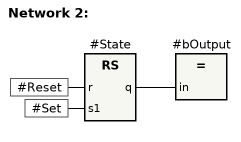
   IF #Reset THEN
       #State := FALSE;   // RS flip-flop
   END_IF;
   IF #Set THEN #State := TRUE; END_IF;
   #bOutput := #State;
END_REGION
END_FUNCTION_BLOCK

FUNCTION_BLOCK "fbLowAlarm"   // FB10, FBD
TITLE = Lightweight version of fbAnalogAlarm with only one limit
{ S7_Optimized_Access := 'TRUE' }
VERSION : 0.1
// stored: AutoNumber true, IsIECCheckEnabled false, IsRetainMemResEnabled false, MemoryReserve 0, SetENOAutomatically false, UDAEnableTagReadback false
   VAR_INPUT
      sValue : "stCalcValue";
      bAckAll : Bool;
      bEnable : Bool;
   END_VAR
   VAR_IN_OUT
      sTag : "stLimitAlarm";
   END_VAR
   VAR
      Alarm : "fbLimitAlarm";
   END_VAR
   VAR CONSTANT
      Low : Bool;
      High : Bool := true;
   END_VAR
BEGIN

REGION Network 1
   // Note that alarm is disabled if CalcValue .bError is set
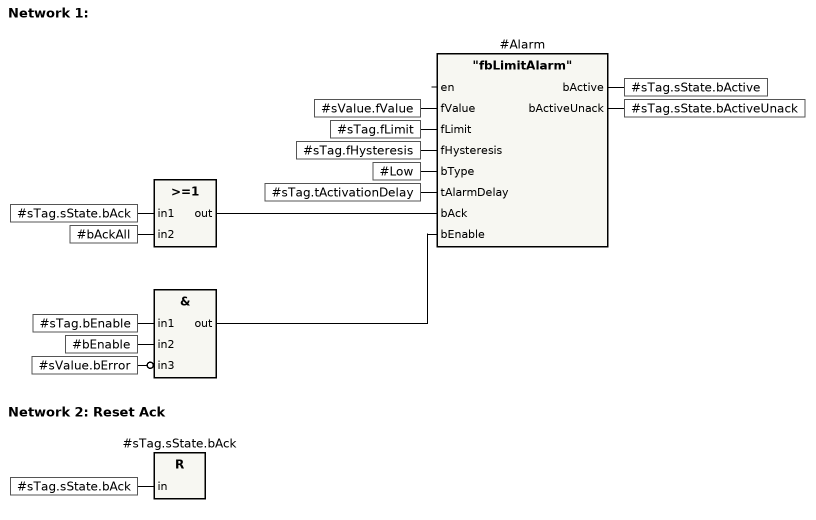
   #Alarm(fValue := #sValue.fValue,   // "fbLimitAlarm"
          fLimit := #sTag.fLimit,
          fHysteresis := #sTag.fHysteresis,
          bType := #Low,
          tAlarmDelay := #sTag.tActivationDelay,
          bAck := #sTag.sState.bAck OR #bAckAll,
          bEnable := #sTag.bEnable AND #bEnable AND NOT #sValue.bError,
          bActive => #sTag.sState.bActive,
          bActiveUnack => #sTag.sState.bActiveUnack);
END_REGION

REGION Network 2: Reset Ack
   IF #sTag.sState.bAck THEN #sTag.sState.bAck := FALSE; END_IF;
END_REGION
END_FUNCTION_BLOCK

FUNCTION_BLOCK "fbDeviationAlarm"   // FB55, FBD
{ S7_Optimized_Access := 'TRUE' }
AUTHOR : Heaten
VERSION : 0.1
// stored: AutoNumber true, IsIECCheckEnabled false, IsRetainMemResEnabled false, MemoryReserve 0, SetENOAutomatically false, UDAEnableTagReadback false
   VAR_INPUT
      sActualValue : "stCalcValue";   // Process value
      fCommandValue : Real;   // Setpoint
      bAckAll : Bool;
      bEnable : Bool;
   END_VAR
   VAR_IN_OUT
      sTag : "stDeviationAlarm";
   END_VAR
   VAR
      Alarm : "fbAlarm";
   END_VAR
   VAR_TEMP
      AlarmCondition : Bool;
   END_VAR
BEGIN

REGION Network 1 (SCL): Alarm condition if measured value ok
   IF #sActualValue.bError = FALSE THEN
       #AlarmCondition := ABS(#sActualValue.fValue - #fCommandValue) > #sTag.fDeviationLimit;
   ELSE
       #AlarmCondition := FALSE;
   END_IF;
END_REGION

REGION Network 2: Alarm with activation delay
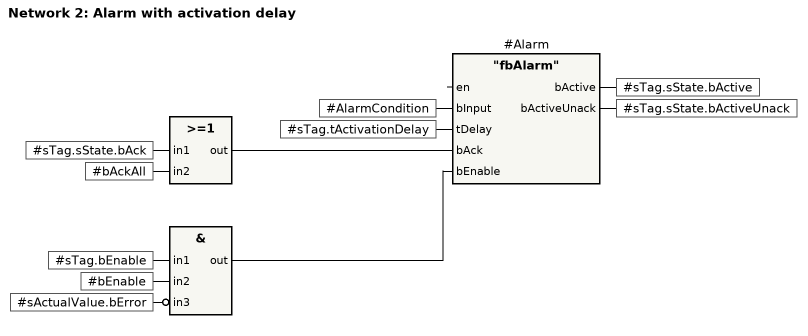
   #Alarm(bInput := #AlarmCondition,   // "fbAlarm"
          tDelay := #sTag.tActivationDelay,
          bAck := #sTag.sState.bAck OR #bAckAll,
          bEnable := #sTag.bEnable AND #bEnable AND NOT #sActualValue.bError,
          bActive => #sTag.sState.bActive,
          bActiveUnack => #sTag.sState.bActiveUnack);
END_REGION
END_FUNCTION_BLOCK

FUNCTION_BLOCK "Regulation"   // FB5, FBD
{ S7_Optimized_Access := 'TRUE' }
VERSION : 0.1
// stored: AutoNumber true, IsIECCheckEnabled true, IsRetainMemResEnabled false, MemoryReserve 10, SetENOAutomatically false, UDAEnableTagReadback false
   VAR
      ExpValveCurrentPressureLimitation : Bool;
      enEmergencyStop { ExternalAccessible := 'False'; ExternalVisible := 'False'; ExternalWritable := 'False'} : Bool;
      CPCPumpRequestFromCPC { ExternalAccessible := 'False'; ExternalVisible := 'False'; ExternalWritable := 'False'} : Bool;   // Crankcase Pressure Control wants to run CPC pump
      CPCPumpRequestFromPurge { ExternalAccessible := 'False'; ExternalVisible := 'False'; ExternalWritable := 'False'} : Bool;   // Do compressor manifold purge
      ExpValveCurrentPressureTarged : Real;
      PerformanceControl_PerformanceRate : Real;
      PerformanceControl { ExternalAccessible := 'False'; ExternalVisible := 'False'; ExternalWritable := 'False'; S7_SetPoint := 'True'} : "PerformanceControl";   // Compressor setpoint
      SuperheatControl { ExternalAccessible := 'False'; ExternalVisible := 'False'; ExternalWritable := 'False'; S7_SetPoint := 'True'} : "SuperheatControl";   // Superheat setpoint
      PinchControl { ExternalAccessible := 'False'; ExternalVisible := 'False'; ExternalWritable := 'False'; S7_SetPoint := 'True'} : "PinchControl";
      CrankcaseOilHeating { ExternalAccessible := 'False'; ExternalVisible := 'False'; ExternalWritable := 'False'; S7_SetPoint := 'True'} : "OilHeating";
      MotorSpeedControl { ExternalAccessible := 'False'; ExternalVisible := 'False'; ExternalWritable := 'False'; S7_SetPoint := 'True'} : "MotorControl";
      SafetyRelay { ExternalAccessible := 'False'; ExternalVisible := 'False'; ExternalWritable := 'False'; S7_SetPoint := 'True'} : "fbSafetyRelay";
      CabinetTemperature { ExternalAccessible := 'False'; ExternalVisible := 'False'; ExternalWritable := 'False'; S7_SetPoint := 'True'} : "fbTemperatureController2";
      ContainerVentilation { ExternalAccessible := 'False'; ExternalVisible := 'False'; ExternalWritable := 'False'; S7_SetPoint := 'True'} : "fbPI_Regulator";
      CrankcasePressureControl { ExternalAccessible := 'False'; ExternalVisible := 'False'; ExternalWritable := 'False'; S7_SetPoint := 'True'} : "CrankcasePressureControl";
      OilSeparator { ExternalAccessible := 'False'; ExternalVisible := 'False'; ExternalWritable := 'False'; S7_SetPoint := 'True'} : "OilSeparator";
      ShaftSealCartridge { ExternalAccessible := 'False'; ExternalVisible := 'False'; ExternalWritable := 'False'; S7_SetPoint := 'True'} : "ShaftSealCartridge";
      LubricationPriming { ExternalAccessible := 'False'; ExternalVisible := 'False'; ExternalWritable := 'False'; S7_SetPoint := 'True'} : "LubricationPriming";
      ValveControl { ExternalAccessible := 'False'; ExternalVisible := 'False'; ExternalWritable := 'False'; S7_SetPoint := 'True'} : "ValveControl";
      PurgeControl { ExternalAccessible := 'False'; ExternalVisible := 'False'; ExternalWritable := 'False'; S7_SetPoint := 'True'} : "fbPurgeControl";
      FilterDryer { S7_SetPoint := 'True'} : "fbFilterDryer";
      OilRecovery { S7_SetPoint := 'True'} : "fbOilRecovery";
      RecuperatorBypass { S7_SetPoint := 'True'} : "fbNullRegulator";
      HeatSourceCycle { S7_SetPoint := 'True'} : "fbTrackingRegulator";
      HeatSourceCyclePIP { S7_SetPoint := 'True'} : "fbPIP_Regulator";
      HeatboosterSetpointPrev { ExternalAccessible := 'False'; ExternalVisible := 'False'; ExternalWritable := 'False'} : Real;   // TEST
      HeatSinkSetpointPrev { ExternalAccessible := 'False'; ExternalVisible := 'False'; ExternalWritable := 'False'} : Real;   // TEST
      HeatSourceSetpointPrev { ExternalAccessible := 'False'; ExternalVisible := 'False'; ExternalWritable := 'False'} : Real;   // TEST
      VariableSetpointPrev { ExternalAccessible := 'False'; ExternalVisible := 'False'; ExternalWritable := 'False'} : Real;
      RegulationTarget { ExternalAccessible := 'False'; ExternalVisible := 'False'; ExternalWritable := 'False'} : Int;   // TEST
      epHeatSinkControlActive { ExternalAccessible := 'False'; ExternalVisible := 'False'; ExternalWritable := 'False'} : Bool;
      epHeatSourceControlActive { ExternalAccessible := 'False'; ExternalVisible := 'False'; ExternalWritable := 'False'} : Bool;
      epVariableControlActive { ExternalAccessible := 'False'; ExternalVisible := 'False'; ExternalWritable := 'False'} : Bool;
      TEST1 : Bool;
   END_VAR
   VAR_TEMP
      AdditionalSuperHeat : Real;
      PerformanceSetpoint : Real;
      AdditionalSuperheatPinch : Real;
   END_VAR
   VAR_TEMP   // added for the SCL form of the ladder/FBD networks
      _w1 : Bool;
   END_VAR
BEGIN

REGION Network 1: Performance control
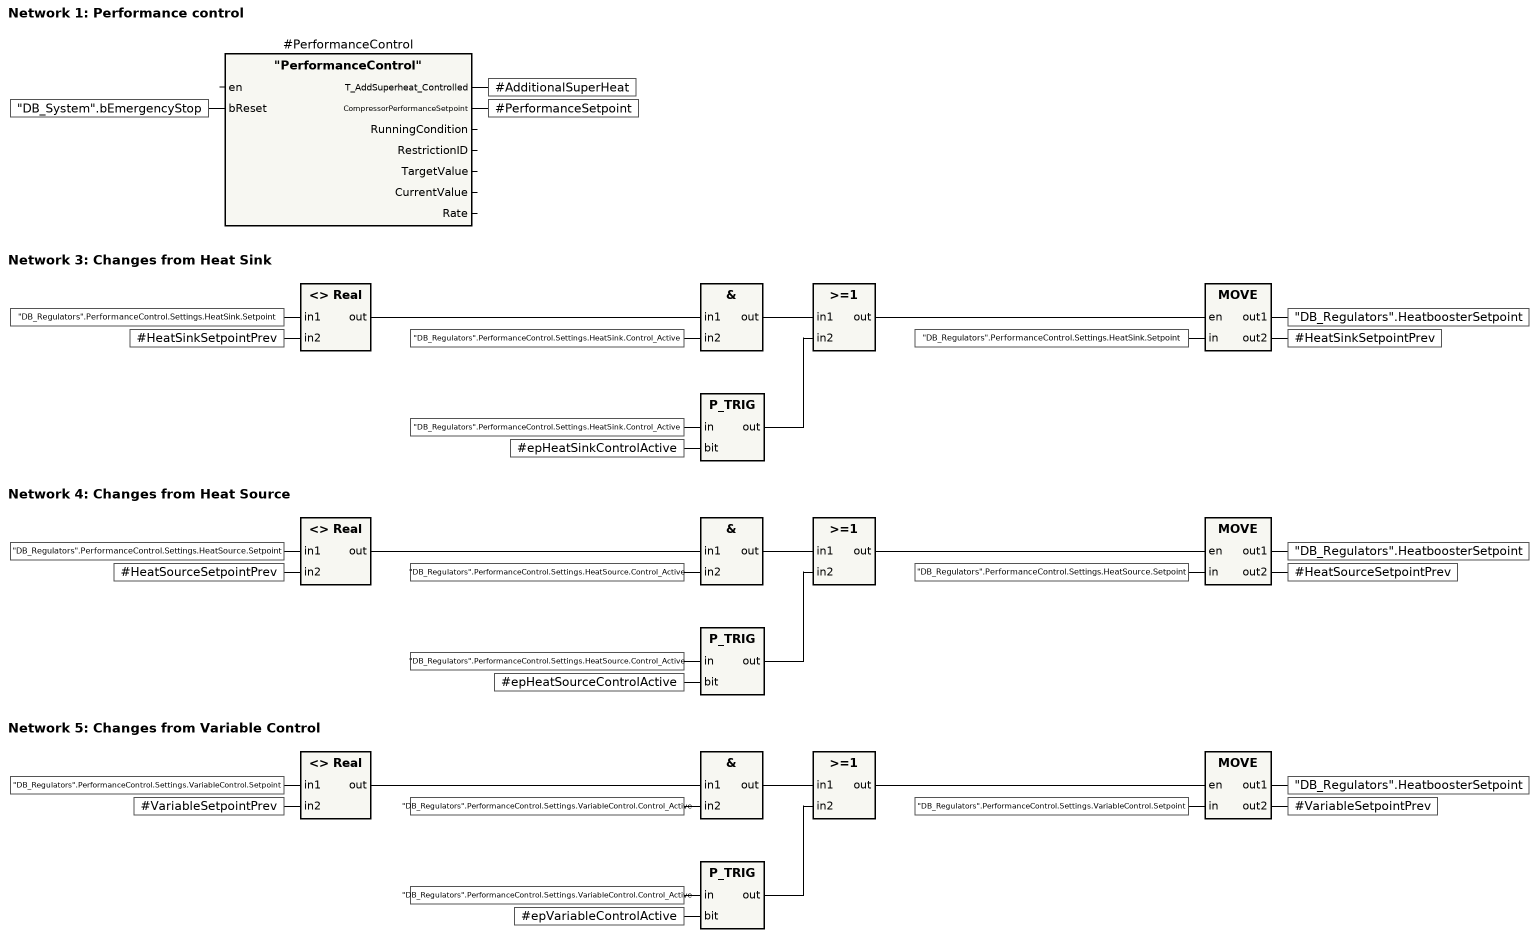
   #PerformanceControl(bReset := "DB_System".bEmergencyStop,   // "PerformanceControl"
                       T_AddSuperheat_Controlled => #AdditionalSuperHeat,
                       CompressorPerformanceSetpoint => #PerformanceSetpoint);
END_REGION

REGION Network 2 (SCL): Performance rate
   // Used in HMI only
   IF "DB_State".State."5_Warmup" OR "DB_State".State."6_Running" AND #PerformanceControl.RunningCondition = TRUE THEN
       #PerformanceControl_PerformanceRate := #MotorSpeedControl.NEngineSetpoint / 15 - #AdditionalSuperHeat / 50 * 30;
   ELSE
       #PerformanceControl_PerformanceRate := 0;
   END_IF;
END_REGION

REGION Network 3: Changes from Heat Sink
   // Propagate setpoint when controller is first activated, or if active and setpoint is changed
   #_w1 := "DB_Regulators".PerformanceControl.Settings.HeatSink.Control_Active AND NOT #epHeatSinkControlActive;   // rising edge
   #epHeatSinkControlActive := "DB_Regulators".PerformanceControl.Settings.HeatSink.Control_Active;
   IF (("DB_Regulators".PerformanceControl.Settings.HeatSink.Setpoint <> #HeatSinkSetpointPrev) AND "DB_Regulators".PerformanceControl.Settings.HeatSink.Control_Active) OR #_w1 THEN
       "DB_Regulators".HeatboosterSetpoint := "DB_Regulators".PerformanceControl.Settings.HeatSink.Setpoint;
       #HeatSinkSetpointPrev := "DB_Regulators".PerformanceControl.Settings.HeatSink.Setpoint;
   END_IF;
END_REGION

REGION Network 4: Changes from Heat Source
   // Propagate setpoint when controller is first activated, or if active and setpoint is changed
   #_w1 := "DB_Regulators".PerformanceControl.Settings.HeatSource.Control_Active AND NOT #epHeatSourceControlActive;   // rising edge
   #epHeatSourceControlActive := "DB_Regulators".PerformanceControl.Settings.HeatSource.Control_Active;
   IF (("DB_Regulators".PerformanceControl.Settings.HeatSource.Setpoint <> #HeatSourceSetpointPrev) AND "DB_Regulators".PerformanceControl.Settings.HeatSource.Control_Active) OR #_w1 THEN
       "DB_Regulators".HeatboosterSetpoint := "DB_Regulators".PerformanceControl.Settings.HeatSource.Setpoint;
       #HeatSourceSetpointPrev := "DB_Regulators".PerformanceControl.Settings.HeatSource.Setpoint;
   END_IF;
END_REGION

REGION Network 5: Changes from Variable Control
   // Propagate setpoint when controller is first activated, or if active and setpoint is changed
   #_w1 := "DB_Regulators".PerformanceControl.Settings.VariableControl.Control_Active AND NOT #epVariableControlActive;   // rising edge
   #epVariableControlActive := "DB_Regulators".PerformanceControl.Settings.VariableControl.Control_Active;
   IF (("DB_Regulators".PerformanceControl.Settings.VariableControl.Setpoint <> #VariableSetpointPrev) AND "DB_Regulators".PerformanceControl.Settings.VariableControl.Control_Active) OR #_w1 THEN
       "DB_Regulators".HeatboosterSetpoint := "DB_Regulators".PerformanceControl.Settings.VariableControl.Setpoint;
       #VariableSetpointPrev := "DB_Regulators".PerformanceControl.Settings.VariableControl.Setpoint;
   END_IF;
END_REGION

REGION Network 6 (SCL): Regulation target
   // No, I didn't suddenly develop a brain hemorrage, this mess here is on purpose:
   // 1. It is a sequence of separate IFs as it mirrors the logic in PerformanceControl
   // 2. It is tempting to re-use Restriction ID, but this can take on values other than the ones here, which we want to avoid. So the value has to be reconstructed.
   // Figure out which target is active
   "DB_Regulators".RegulationTarget := 0;  // in case none of the regulators are active, none of the IFs fire...
   IF "DB_Regulators".PerformanceControl.Settings.HeatSink.Control_Active THEN
       IF "DB_Regulators".PerformanceControl.Settings.HeatSink.UseFeedFlow THEN
           "DB_Regulators".RegulationTarget := 2;
       ELSE
           "DB_Regulators".RegulationTarget := 1;
       END_IF;
   END_IF;

   IF "DB_Regulators".PerformanceControl.Settings.HeatSource.Control_Active THEN
       IF "DB_Regulators".PerformanceControl.Settings.HeatSource.UseFeedFlow THEN
           "DB_Regulators".RegulationTarget := 4;
       ELSE
           "DB_Regulators".RegulationTarget := 3;
       END_IF;
   END_IF;

   IF "DB_Regulators".PerformanceControl.Settings.VariableControl.Control_Active AND "DB_Regulators".PerformanceControl.Settings.VariableControl.ReferenceID > 0 THEN
       "DB_Regulators".RegulationTarget := 6;
   END_IF;
END_REGION

REGION Network 7: Changes from DB_Regulators
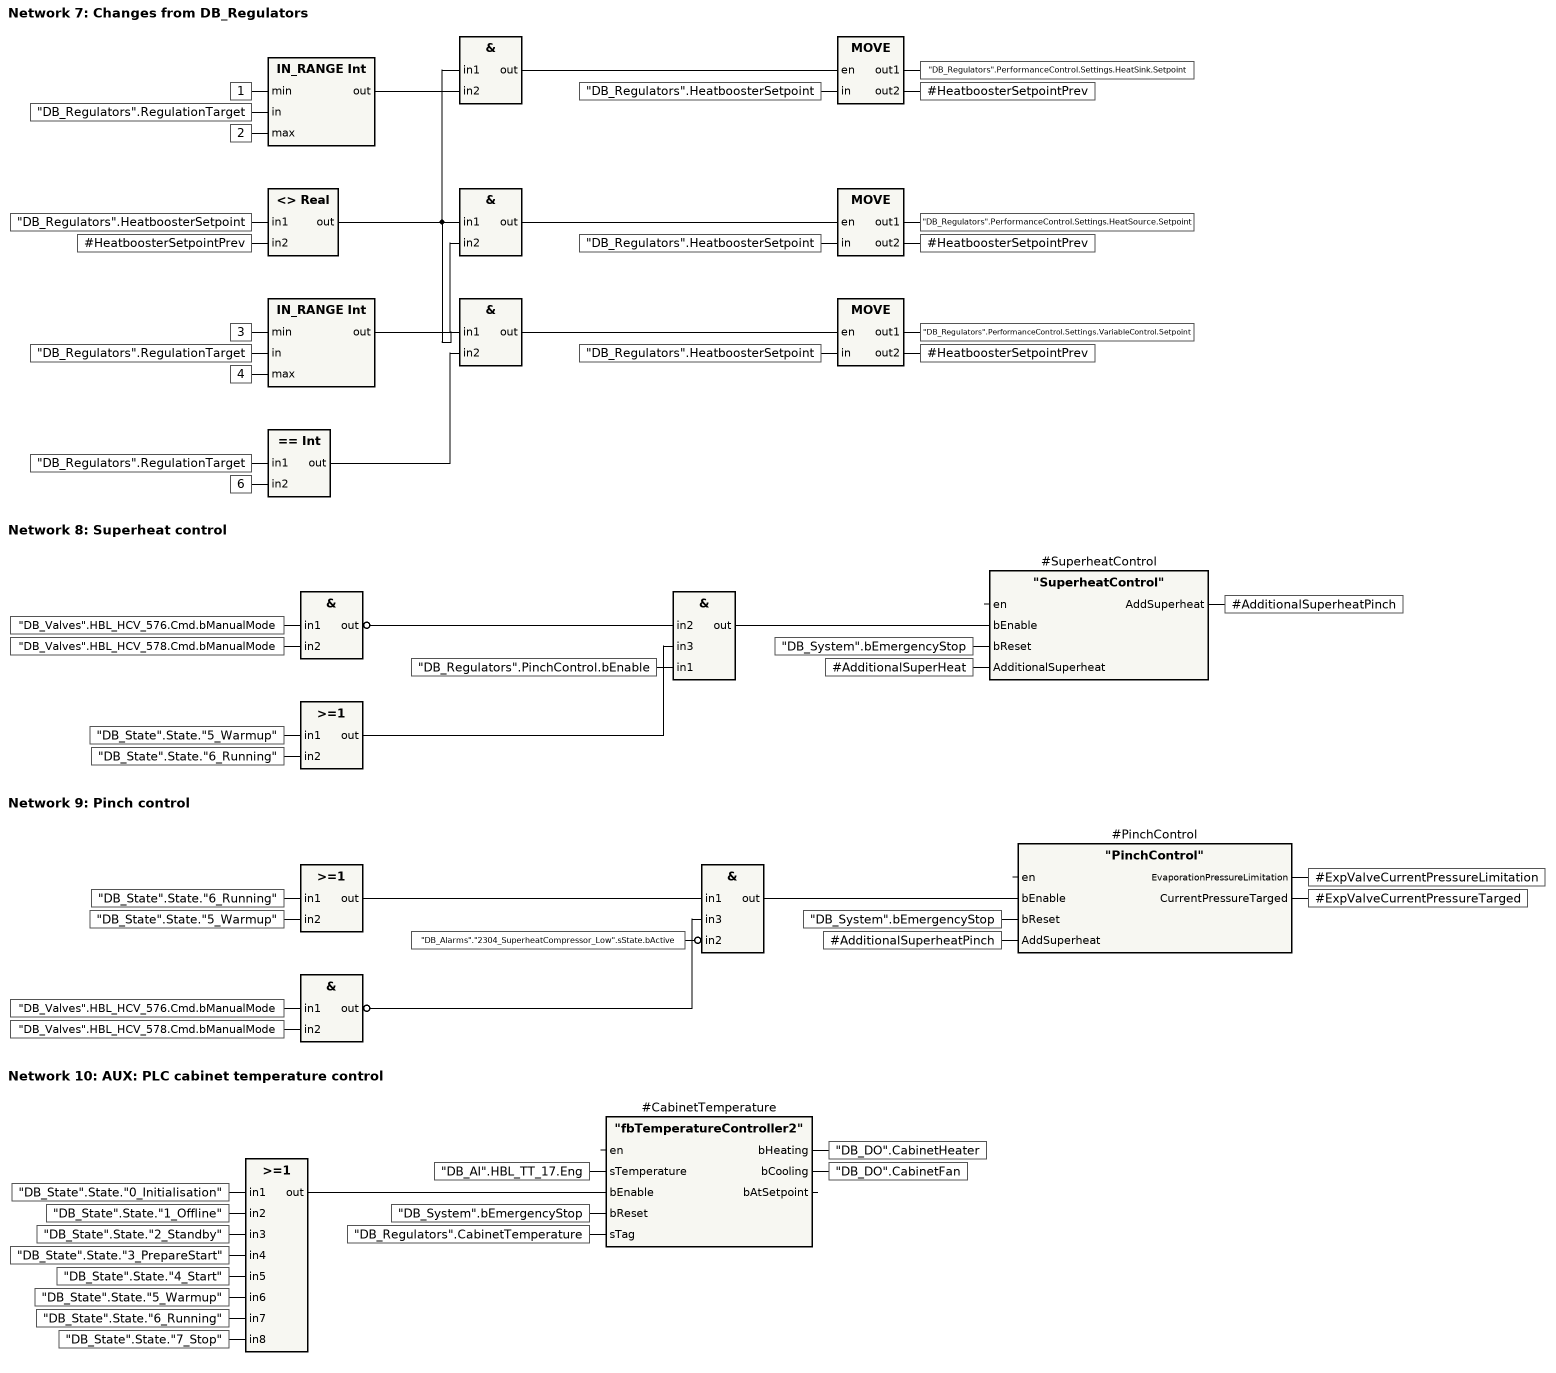
   #_w1 := "DB_Regulators".HeatboosterSetpoint <> #HeatboosterSetpointPrev;
   IF #_w1 AND (1 <= "DB_Regulators".RegulationTarget) AND ("DB_Regulators".RegulationTarget <= 2) THEN
       "DB_Regulators".PerformanceControl.Settings.HeatSink.Setpoint := "DB_Regulators".HeatboosterSetpoint;
       #HeatboosterSetpointPrev := "DB_Regulators".HeatboosterSetpoint;
   END_IF;
   IF #_w1 AND (3 <= "DB_Regulators".RegulationTarget) AND ("DB_Regulators".RegulationTarget <= 4) THEN
       "DB_Regulators".PerformanceControl.Settings.HeatSource.Setpoint := "DB_Regulators".HeatboosterSetpoint;
       #HeatboosterSetpointPrev := "DB_Regulators".HeatboosterSetpoint;
   END_IF;
   IF #_w1 AND ("DB_Regulators".RegulationTarget = 6) THEN
       "DB_Regulators".PerformanceControl.Settings.VariableControl.Setpoint := "DB_Regulators".HeatboosterSetpoint;
       #HeatboosterSetpointPrev := "DB_Regulators".HeatboosterSetpoint;
   END_IF;
END_REGION

REGION Network 8: Superheat control
   #SuperheatControl(bEnable := NOT ("DB_Valves".HBL_HCV_576.Cmd.bManualMode AND "DB_Valves".HBL_HCV_578.Cmd.bManualMode) AND ("DB_State".State."5_Warmup" OR "DB_State".State."6_Running") AND "DB_Regulators".PinchControl.bEnable,   // "SuperheatControl"
                     bReset := "DB_System".bEmergencyStop,
                     AdditionalSuperheat := #AdditionalSuperHeat,
                     AddSuperheat => #AdditionalSuperheatPinch);
END_REGION

REGION Network 9: Pinch control
   #PinchControl(bEnable := ("DB_State".State."6_Running" OR "DB_State".State."5_Warmup") AND NOT ("DB_Valves".HBL_HCV_576.Cmd.bManualMode AND "DB_Valves".HBL_HCV_578.Cmd.bManualMode) AND NOT "DB_Alarms"."2304_SuperheatCompressor_Low".sState.bActive,   // "PinchControl"
                 bReset := "DB_System".bEmergencyStop,
                 AddSuperheat := #AdditionalSuperheatPinch,
                 EvaporationPressureLimitation => #ExpValveCurrentPressureLimitation,
                 CurrentPressureTarged => #ExpValveCurrentPressureTarged);
END_REGION

REGION Network 10: AUX: PLC cabinet temperature control
   // Runs all the time, as the cabinet is running all the time...
   #CabinetTemperature(sTemperature := "DB_AI".HBL_TT_17.Eng,   // "fbTemperatureController2"
                       bEnable := "DB_State".State."0_Initialisation" OR "DB_State".State."1_Offline" OR "DB_State".State."2_Standby" OR "DB_State".State."3_PrepareStart" OR "DB_State".State."4_Start" OR "DB_State".State."5_Warmup" OR "DB_State".State."6_Running" OR "DB_State".State."7_Stop",
                       bReset := "DB_System".bEmergencyStop,
                       sTag := "DB_Regulators".CabinetTemperature,
                       bHeating => "DB_DO".CabinetHeater,
                       bCooling => "DB_DO".CabinetFan);
END_REGION

REGION Network 11: AUX: Crankcase oil heater control
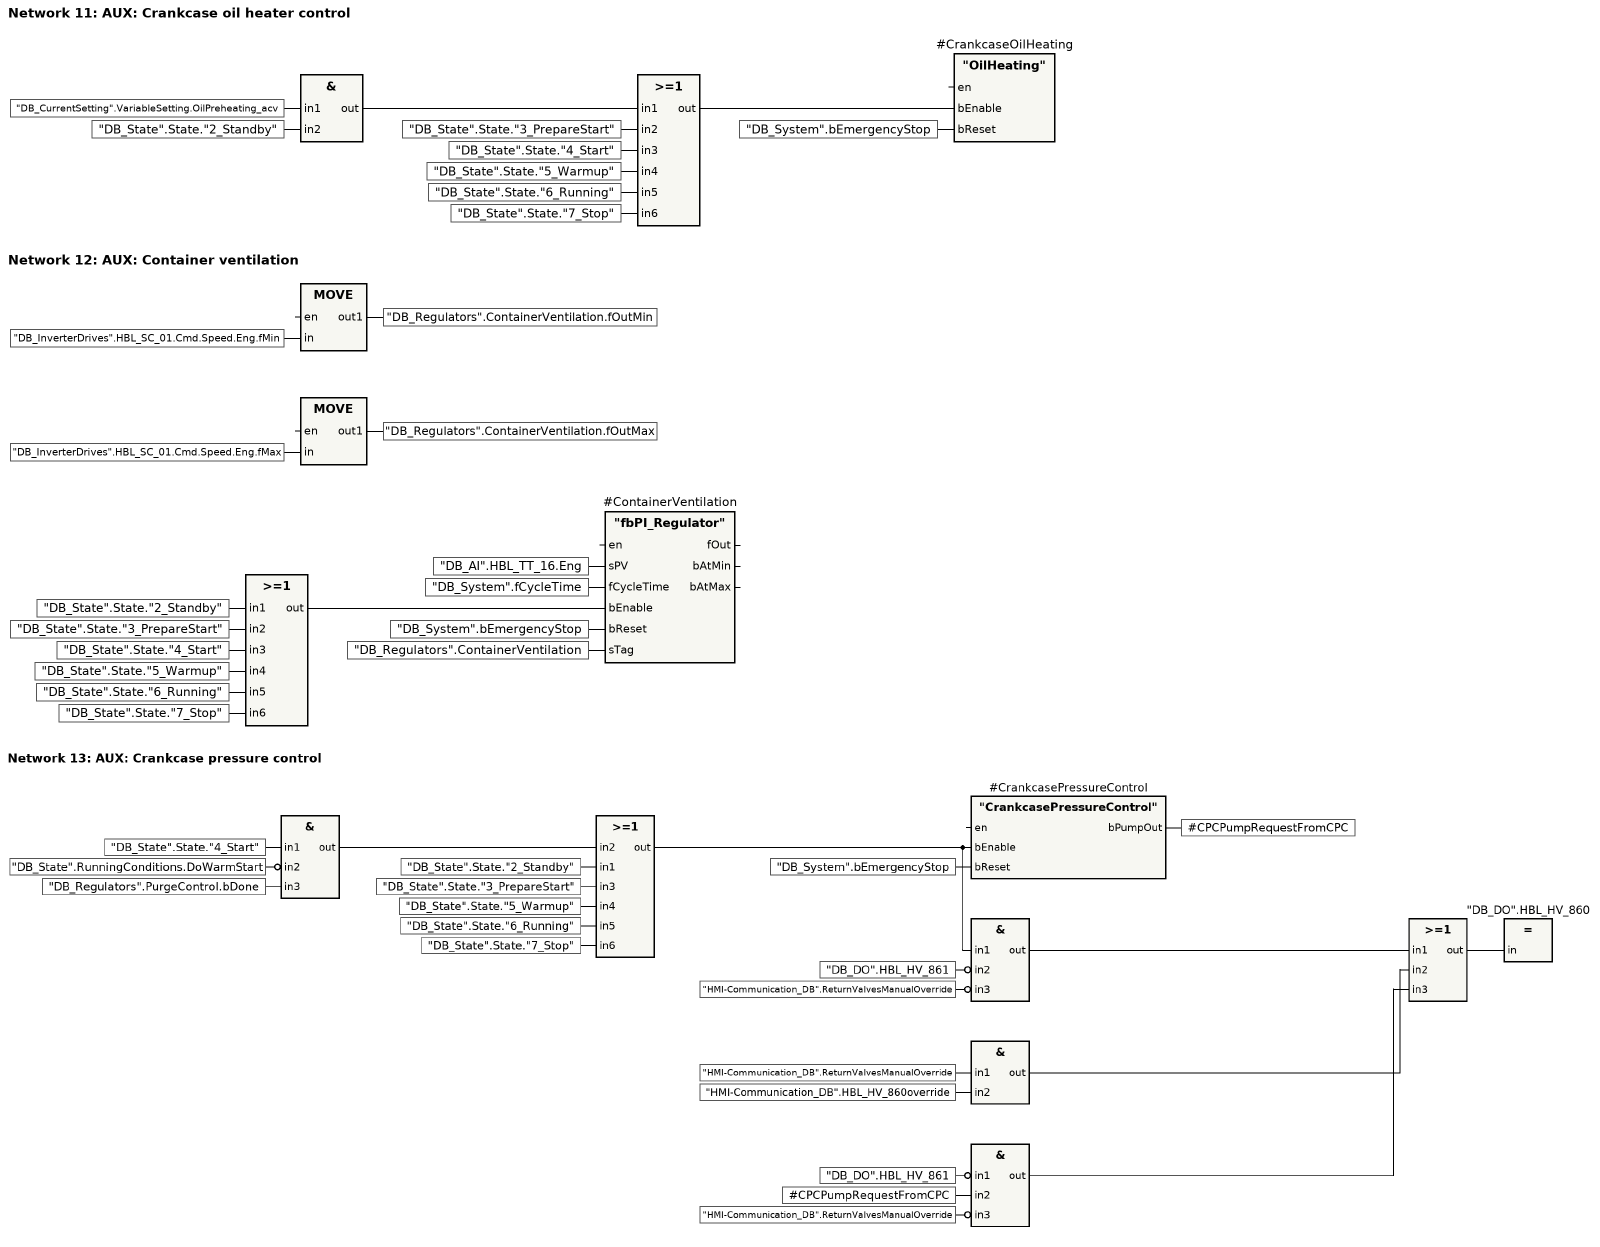
   #CrankcaseOilHeating(bEnable := ("DB_CurrentSetting".VariableSetting.OilPreheating_acv AND "DB_State".State."2_Standby") OR "DB_State".State."3_PrepareStart" OR "DB_State".State."4_Start" OR "DB_State".State."5_Warmup" OR "DB_State".State."6_Running" OR "DB_State".State."7_Stop",   // "OilHeating"
                        bReset := "DB_System".bEmergencyStop);
END_REGION

REGION Network 12: AUX: Container ventilation
   // Manually copy the actuator min & max to the regulator min & max. This is not automatically true for all regulators
   // ##FIX: Hack the start signal, ugliness alert
   "DB_Regulators".ContainerVentilation.fOutMin := "DB_InverterDrives".HBL_SC_01.Cmd.Speed.Eng.fMin;
   "DB_Regulators".ContainerVentilation.fOutMax := "DB_InverterDrives".HBL_SC_01.Cmd.Speed.Eng.fMax;
   #ContainerVentilation(sPV := "DB_AI".HBL_TT_16.Eng,   // "fbPI_Regulator"
                         fCycleTime := "DB_System".fCycleTime,
                         bEnable := "DB_State".State."2_Standby" OR "DB_State".State."3_PrepareStart" OR "DB_State".State."4_Start" OR "DB_State".State."5_Warmup" OR "DB_State".State."6_Running" OR "DB_State".State."7_Stop",
                         bReset := "DB_System".bEmergencyStop,
                         sTag := "DB_Regulators".ContainerVentilation);
END_REGION

REGION Network 13: AUX: Crankcase pressure control
   // Disable the controller temporarily in State 4 Start when doing a cold start
   #_w1 := ("DB_State".State."4_Start" AND NOT "DB_State".RunningConditions.DoWarmStart AND "DB_Regulators".PurgeControl.bDone) OR "DB_State".State."2_Standby" OR "DB_State".State."3_PrepareStart" OR "DB_State".State."5_Warmup" OR "DB_State".State."6_Running" OR "DB_State".State."7_Stop";
   #CrankcasePressureControl(bEnable := #_w1,   // "CrankcasePressureControl"
                           bReset := "DB_System".bEmergencyStop,
                           bPumpOut => #CPCPumpRequestFromCPC);
   "DB_DO".HBL_HV_860 := (#_w1 AND NOT "DB_DO".HBL_HV_861 AND NOT "HMI-Communication_DB".ReturnValvesManualOverride) OR ("HMI-Communication_DB".ReturnValvesManualOverride AND "HMI-Communication_DB".HBL_HV_860override) OR (NOT "DB_DO".HBL_HV_861 AND #CPCPumpRequestFromCPC AND NOT "HMI-Communication_DB".ReturnValvesManualOverride);
END_REGION

REGION Network 14: AUX: Oil separator level control
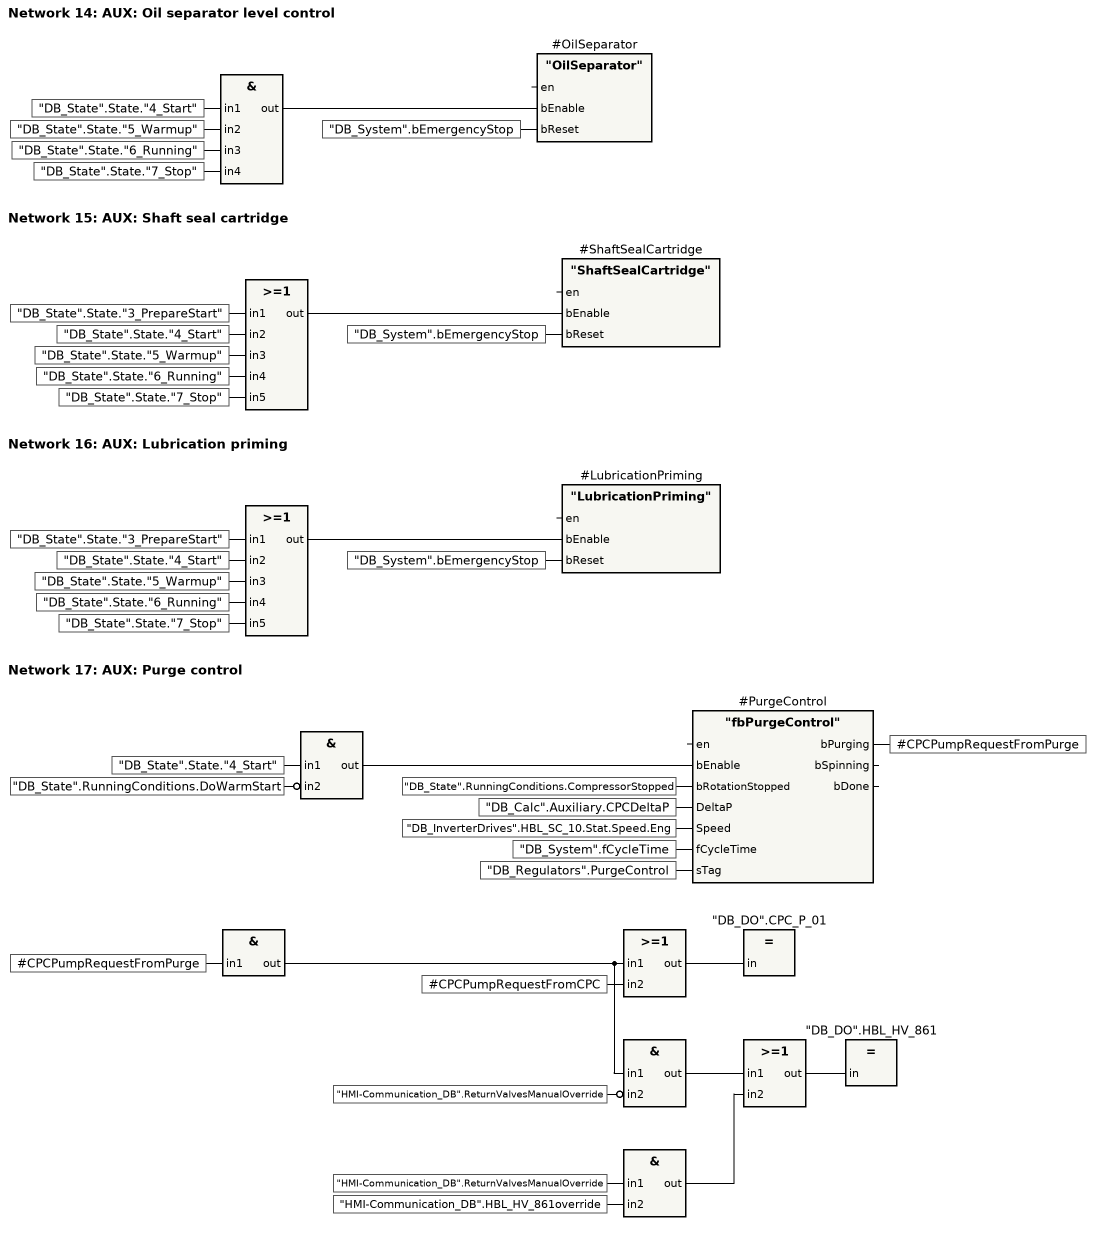
   #OilSeparator(bEnable := "DB_State".State."4_Start" AND "DB_State".State."5_Warmup" AND "DB_State".State."6_Running" AND "DB_State".State."7_Stop",   // "OilSeparator"
                 bReset := "DB_System".bEmergencyStop);
END_REGION

REGION Network 15: AUX: Shaft seal cartridge
   #ShaftSealCartridge(bEnable := "DB_State".State."3_PrepareStart" OR "DB_State".State."4_Start" OR "DB_State".State."5_Warmup" OR "DB_State".State."6_Running" OR "DB_State".State."7_Stop",   // "ShaftSealCartridge"
                       bReset := "DB_System".bEmergencyStop);
END_REGION

REGION Network 16: AUX: Lubrication priming
   #LubricationPriming(bEnable := "DB_State".State."3_PrepareStart" OR "DB_State".State."4_Start" OR "DB_State".State."5_Warmup" OR "DB_State".State."6_Running" OR "DB_State".State."7_Stop",   // "LubricationPriming"
                       bReset := "DB_System".bEmergencyStop);
END_REGION

REGION Network 17: AUX: Purge control
   // Note: HBL-XV-05 takes priority over HBL-XV-04
   #PurgeControl(bEnable := "DB_State".State."4_Start" AND NOT "DB_State".RunningConditions.DoWarmStart,   // "fbPurgeControl"
                 bRotationStopped := "DB_State".RunningConditions.CompressorStopped,
                 DeltaP := "DB_Calc".Auxiliary.CPCDeltaP,
                 Speed := "DB_InverterDrives".HBL_SC_10.Stat.Speed.Eng,
                 fCycleTime := "DB_System".fCycleTime,
                 sTag := "DB_Regulators".PurgeControl,
                 bPurging => #CPCPumpRequestFromPurge);
   "DB_DO".CPC_P_01 := #CPCPumpRequestFromPurge OR #CPCPumpRequestFromCPC;
   "DB_DO".HBL_HV_861 := (#CPCPumpRequestFromPurge AND NOT "HMI-Communication_DB".ReturnValvesManualOverride) OR ("HMI-Communication_DB".ReturnValvesManualOverride AND "HMI-Communication_DB".HBL_HV_861override);
END_REGION

REGION Network 18: AUX: Compressor manifold oil return
   // This is still up in the air what this will be
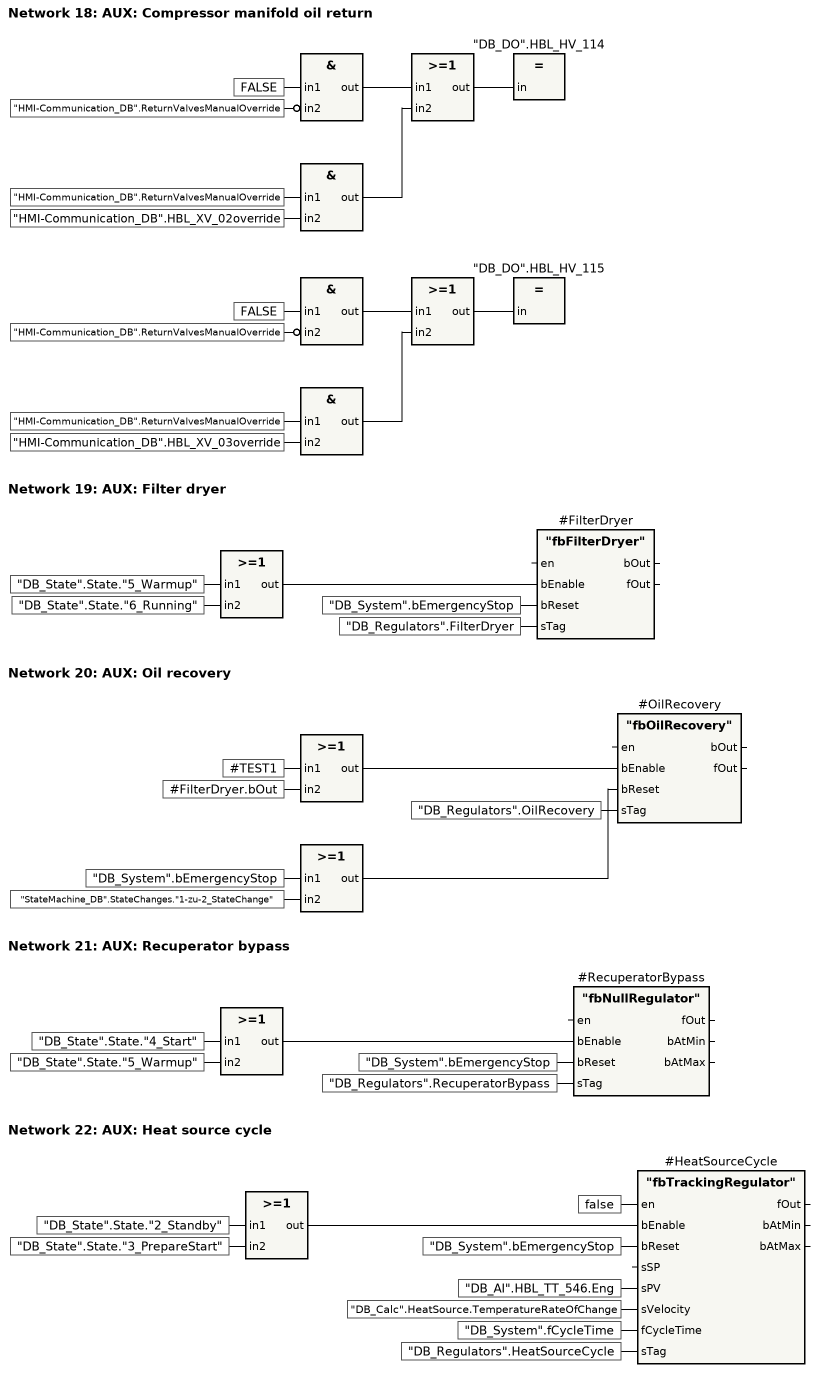
   "DB_DO".HBL_HV_114 := (FALSE AND NOT "HMI-Communication_DB".ReturnValvesManualOverride) OR ("HMI-Communication_DB".ReturnValvesManualOverride AND "HMI-Communication_DB".HBL_XV_02override);
   "DB_DO".HBL_HV_115 := (FALSE AND NOT "HMI-Communication_DB".ReturnValvesManualOverride) OR ("HMI-Communication_DB".ReturnValvesManualOverride AND "HMI-Communication_DB".HBL_XV_03override);
END_REGION

REGION Network 19: AUX: Filter dryer
   #FilterDryer(bEnable := "DB_State".State."5_Warmup" OR "DB_State".State."6_Running",   // "fbFilterDryer"
                bReset := "DB_System".bEmergencyStop,
                sTag := "DB_Regulators".FilterDryer);
END_REGION

REGION Network 20: AUX: Oil recovery
   // Run only when filter dryer is also running
   #OilRecovery(bEnable := #TEST1 OR #FilterDryer.bOut,   // "fbOilRecovery"
                bReset := "DB_System".bEmergencyStop OR "StateMachine_DB".StateChanges."1-zu-2_StateChange",
                sTag := "DB_Regulators".OilRecovery);
END_REGION

REGION Network 21: AUX: Recuperator bypass
   #RecuperatorBypass(bEnable := "DB_State".State."4_Start" OR "DB_State".State."5_Warmup",   // "fbNullRegulator"
                      bReset := "DB_System".bEmergencyStop,
                      sTag := "DB_Regulators".RecuperatorBypass);
END_REGION

REGION Network 22: AUX: Heat source cycle
   IF false THEN
       #HeatSourceCycle(bEnable := "DB_State".State."2_Standby" OR "DB_State".State."3_PrepareStart",   // "fbTrackingRegulator"
                        bReset := "DB_System".bEmergencyStop,
                        sPV := "DB_AI".HBL_TT_546.Eng,
                        sVelocity := "DB_Calc".HeatSource.TemperatureRateOfChange,
                        fCycleTime := "DB_System".fCycleTime,
                        sTag := "DB_Regulators".HeatSourceCycle);
   END_IF;
END_REGION

REGION Network 23: AUX: Heat source cycle PIP
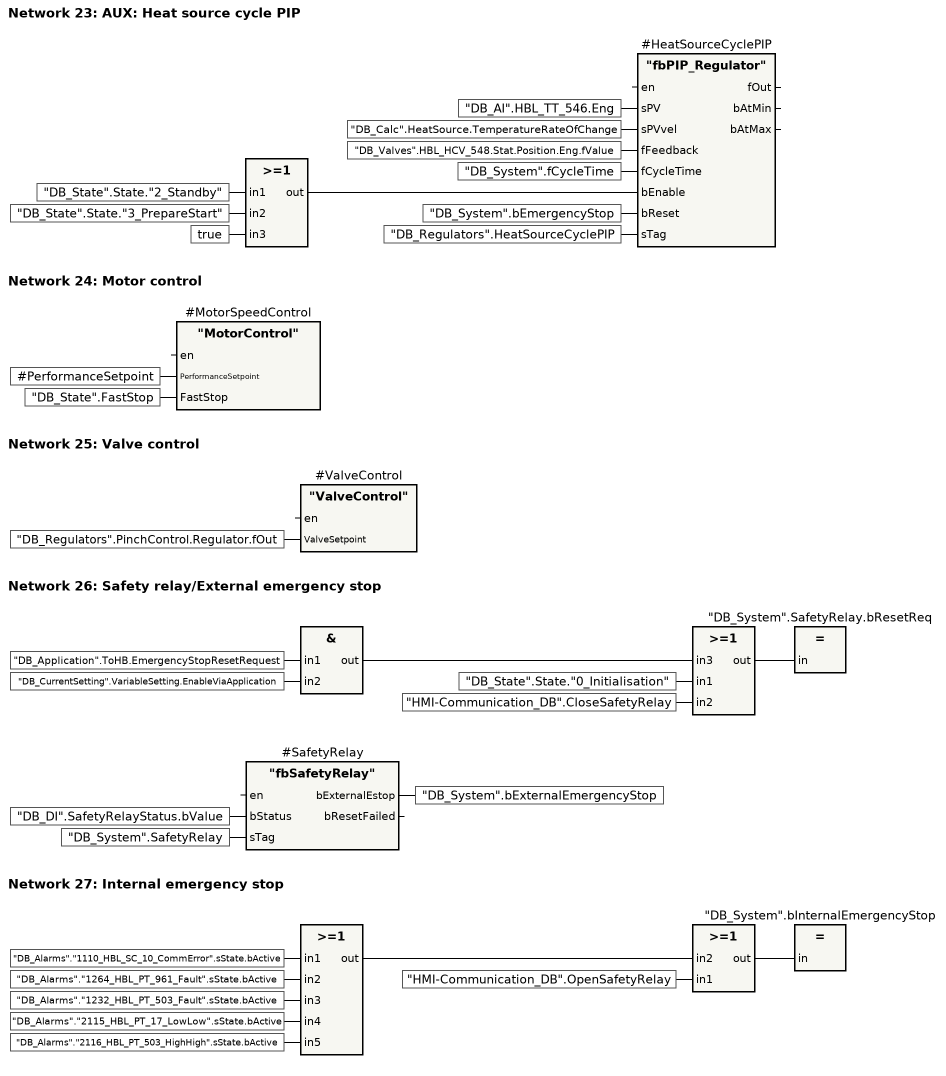
   #HeatSourceCyclePIP(sPV := "DB_AI".HBL_TT_546.Eng,   // "fbPIP_Regulator"
                       sPVvel := "DB_Calc".HeatSource.TemperatureRateOfChange,
                       fFeedback := "DB_Valves".HBL_HCV_548.Stat.Position.Eng.fValue,
                       fCycleTime := "DB_System".fCycleTime,
                       bEnable := "DB_State".State."2_Standby" OR "DB_State".State."3_PrepareStart" OR true,
                       bReset := "DB_System".bEmergencyStop,
                       sTag := "DB_Regulators".HeatSourceCyclePIP);
END_REGION

REGION Network 24: Motor control
   // Note this has to come after all regulators which set the motor speed
   #MotorSpeedControl(PerformanceSetpoint := #PerformanceSetpoint, FastStop := "DB_State".FastStop);   // "MotorControl"
END_REGION

REGION Network 25: Valve control
   #ValveControl(ValveSetpoint := "DB_Regulators".PinchControl.Regulator.fOut);   // "ValveControl"
END_REGION

REGION Network 26: Safety relay/External emergency stop
   "DB_System".SafetyRelay.bResetReq := ("DB_Application".ToHB.EmergencyStopResetRequest AND "DB_CurrentSetting".VariableSetting.EnableViaApplication) OR "DB_State".State."0_Initialisation" OR "HMI-Communication_DB".CloseSafetyRelay;
   #SafetyRelay(bStatus := "DB_DI".SafetyRelayStatus.bValue,   // "fbSafetyRelay"
                sTag := "DB_System".SafetyRelay,
                bExternalEstop => "DB_System".bExternalEmergencyStop);
END_REGION

REGION Network 27: Internal emergency stop
   // The alarms in this list should also be in the Critical alarms list in FB32 AlarmManagement.
   // HBL-PT-17 : lubrication failure, stop compressor (or fault in this sensor)
   // HBL-PT-503: compressor discharge overpressure, stop the compressor (or fault in this sensor)
   // HBL-SC-10: compressor inverter communication loss, no other way to shut it down except by hardwired emergency stop.
   "DB_System".bInternalEmergencyStop := "DB_Alarms"."1110_HBL_SC_10_CommError".sState.bActive OR "DB_Alarms"."1264_HBL_PT_961_Fault".sState.bActive OR "DB_Alarms"."1232_HBL_PT_503_Fault".sState.bActive OR "DB_Alarms"."2115_HBL_PT_17_LowLow".sState.bActive OR "DB_Alarms"."2116_HBL_PT_503_HighHigh".sState.bActive OR "HMI-Communication_DB".OpenSafetyRelay;
END_REGION

REGION Network 28: Emergency stop
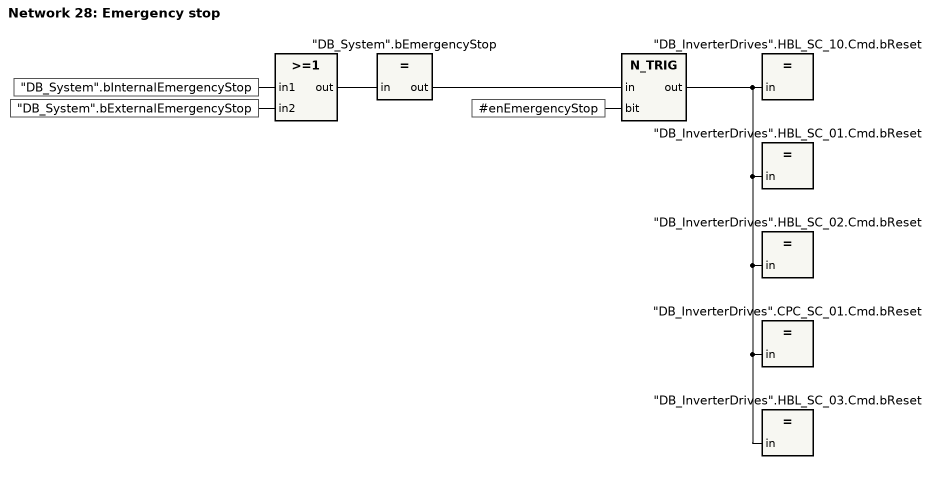
   "DB_System".bEmergencyStop := "DB_System".bInternalEmergencyStop OR "DB_System".bExternalEmergencyStop;
   #_w1 := NOT "DB_System".bEmergencyStop AND #enEmergencyStop;   // falling edge
   #enEmergencyStop := "DB_System".bEmergencyStop;
   "DB_InverterDrives".HBL_SC_10.Cmd.bReset := #_w1;
   "DB_InverterDrives".HBL_SC_01.Cmd.bReset := #_w1;
   "DB_InverterDrives".HBL_SC_02.Cmd.bReset := #_w1;
   "DB_InverterDrives".CPC_SC_01.Cmd.bReset := #_w1;
   "DB_InverterDrives".HBL_SC_03.Cmd.bReset := #_w1;
END_REGION

REGION Network 29: Manual mode warning
   // One or more regulators or actuators is in manual mode.
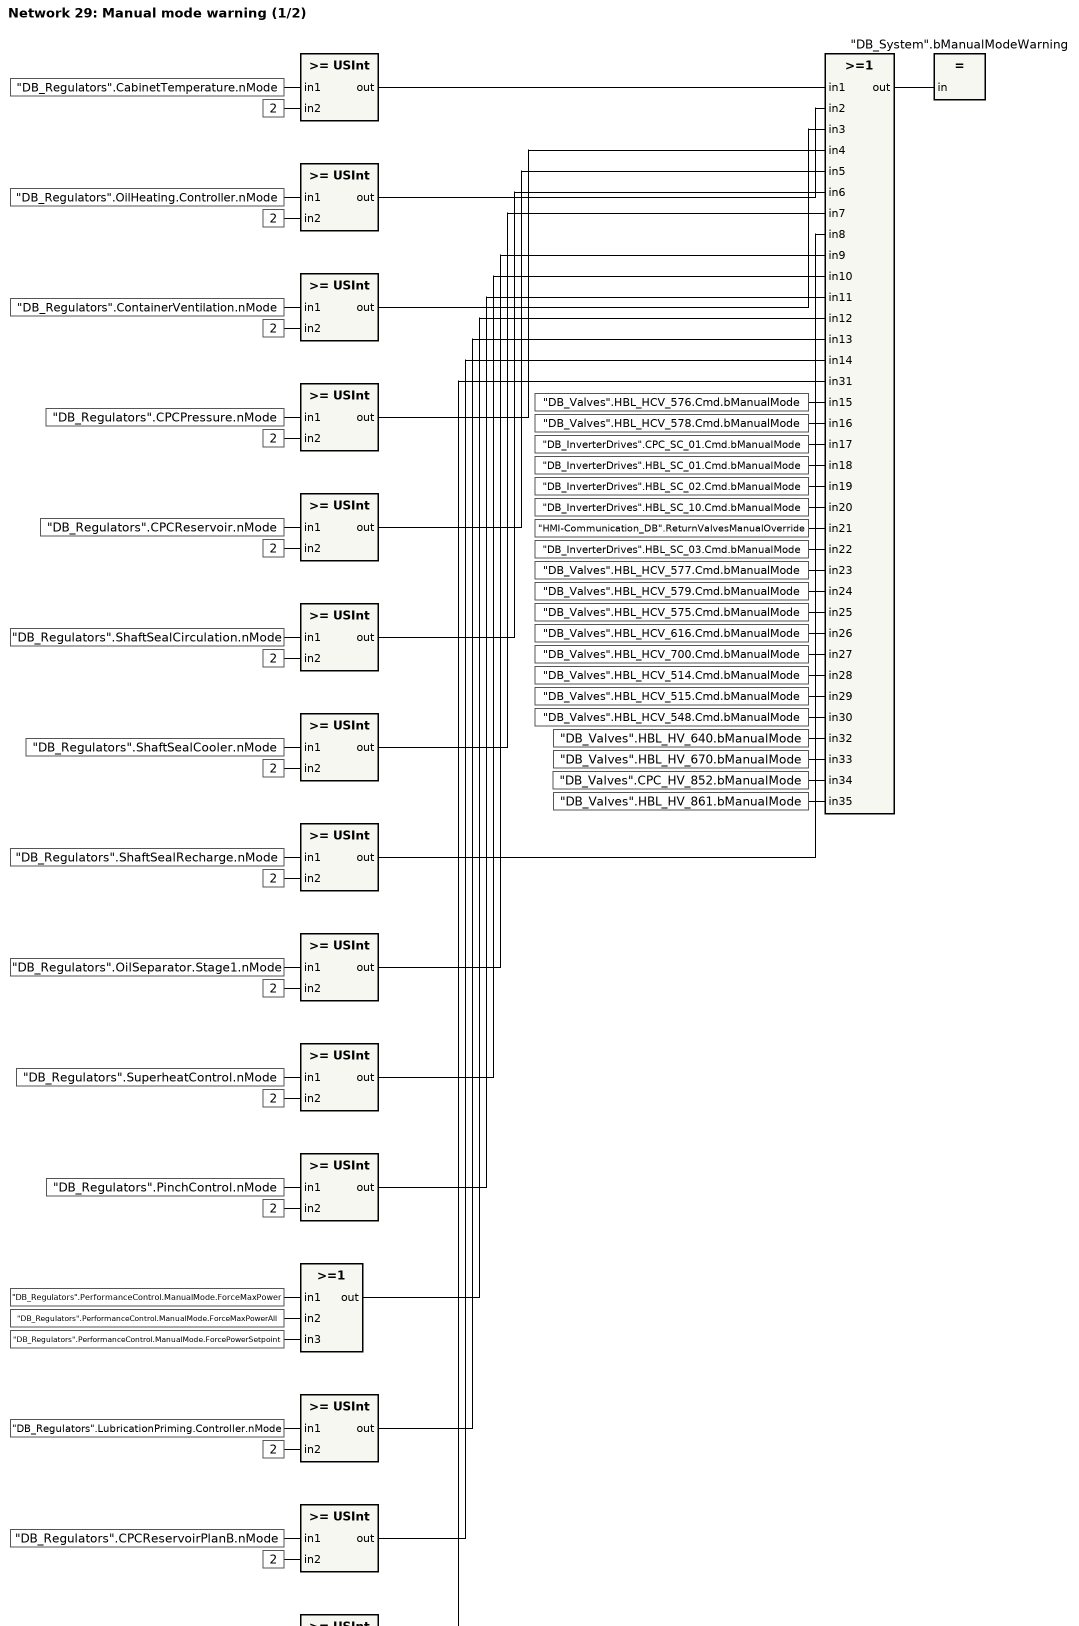
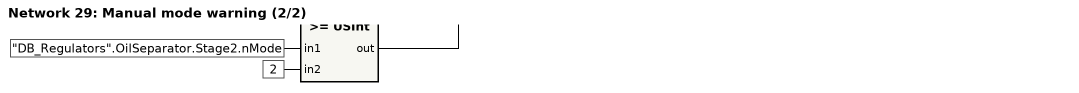
   "DB_System".bManualModeWarning := ("DB_Regulators".CabinetTemperature.nMode >= 2) OR ("DB_Regulators".OilHeating.Controller.nMode >= 2) OR ("DB_Regulators".ContainerVentilation.nMode >= 2) OR ("DB_Regulators".CPCPressure.nMode >= 2) OR ("DB_Regulators".CPCReservoir.nMode >= 2) OR ("DB_Regulators".ShaftSealCirculation.nMode >= 2) OR ("DB_Regulators".ShaftSealCooler.nMode >= 2) OR ("DB_Regulators".ShaftSealRecharge.nMode >= 2) OR ("DB_Regulators".OilSeparator.Stage1.nMode >= 2) OR ("DB_Regulators".SuperheatControl.nMode >= 2) OR ("DB_Regulators".PinchControl.nMode >= 2) OR "DB_Regulators".PerformanceControl.ManualMode.ForceMaxPower OR "DB_Regulators".PerformanceControl.ManualMode.ForceMaxPowerAll OR "DB_Regulators".PerformanceControl.ManualMode.ForcePowerSetpoint OR ("DB_Regulators".LubricationPriming.Controller.nMode >= 2) OR ("DB_Regulators".CPCReservoirPlanB.nMode >= 2) OR ("DB_Regulators".OilSeparator.Stage2.nMode >= 2) OR "DB_Valves".HBL_HCV_576.Cmd.bManualMode OR "DB_Valves".HBL_HCV_578.Cmd.bManualMode OR "DB_InverterDrives".CPC_SC_01.Cmd.bManualMode OR "DB_InverterDrives".HBL_SC_01.Cmd.bManualMode OR "DB_InverterDrives".HBL_SC_02.Cmd.bManualMode OR "DB_InverterDrives".HBL_SC_10.Cmd.bManualMode OR "HMI-Communication_DB".ReturnValvesManualOverride OR "DB_InverterDrives".HBL_SC_03.Cmd.bManualMode OR "DB_Valves".HBL_HCV_577.Cmd.bManualMode OR "DB_Valves".HBL_HCV_579.Cmd.bManualMode OR "DB_Valves".HBL_HCV_575.Cmd.bManualMode OR "DB_Valves".HBL_HCV_616.Cmd.bManualMode OR "DB_Valves".HBL_HCV_700.Cmd.bManualMode OR "DB_Valves".HBL_HCV_514.Cmd.bManualMode OR "DB_Valves".HBL_HCV_515.Cmd.bManualMode OR "DB_Valves".HBL_HCV_548.Cmd.bManualMode OR "DB_Valves".HBL_HV_640.bManualMode OR "DB_Valves".HBL_HV_670.bManualMode OR "DB_Valves".CPC_HV_852.bManualMode OR "DB_Valves".HBL_HV_861.bManualMode;
END_REGION
END_FUNCTION_BLOCK

FUNCTION_BLOCK "PerformanceControl"   // FB9, FBD
TITLE = Performance control
{ S7_Optimized_Access := 'TRUE' }
VERSION : 0.1
// POWER Restiction IDs:
//   1: Customer: Heat sink suction temperature
//   2: Customer: Heat source discharge temperature
//   3: Customer: Heat sink discharge temperature
//   4: Customer: Heat source suction temperature
//   5: Customer: Reserve Analog In
//   6: Customer: Variable control
//   7: Customer: Reserve
//   8: Safety: Safety limit condensing pressure
//   9: Safety: Safety limit compressor motor torque
// 10: Safety: Safety limit compressor motor winding temperature
// 11: Safety: Safety limit container air temperature
// 12: Safety: Safety limit control cabinet air temperature
// 13: Safety: Safety limit compressor inverter temperature
// 14: Safety: Safety limit oil sump oil temperature
// stored: AutoNumber true, IsIECCheckEnabled false, IsRetainMemResEnabled false, MemoryReserve 100, SetENOAutomatically false, UDAEnableTagReadback false
   VAR_INPUT
      bReset { ExternalAccessible := 'False'; ExternalVisible := 'False'; ExternalWritable := 'False'} : Bool;
   END_VAR
   VAR_OUTPUT
      T_AddSuperheat_Controlled { ExternalAccessible := 'False'; ExternalVisible := 'False'; ExternalWritable := 'False'} : Real;
      CompressorPerformanceSetpoint { ExternalAccessible := 'False'; ExternalVisible := 'False'; ExternalWritable := 'False'} : Real;
      RunningCondition { ExternalAccessible := 'False'; ExternalVisible := 'False'; ExternalWritable := 'False'} : Bool;
      RestrictionID { ExternalAccessible := 'False'; ExternalVisible := 'False'; ExternalWritable := 'False'} : Int;
      TargetValue { ExternalAccessible := 'False'; ExternalVisible := 'False'; ExternalWritable := 'False'} : Real;
      CurrentValue { ExternalAccessible := 'False'; ExternalVisible := 'False'; ExternalWritable := 'False'} : Real;
      Rate { ExternalAccessible := 'False'; ExternalVisible := 'False'; ExternalWritable := 'False'} : Real;
   END_VAR
   VAR
      PerformanceRate { ExternalAccessible := 'False'; ExternalVisible := 'False'; ExternalWritable := 'False'} : Real;
      LastDT1_Memory_n { ExternalAccessible := 'False'; ExternalVisible := 'False'; ExternalWritable := 'False'} : Real;
      IntegralPart_Memory_n { ExternalAccessible := 'False'; ExternalVisible := 'False'; ExternalWritable := 'False'} : Real;
      ParameterChange_Memory_n { ExternalAccessible := 'False'; ExternalVisible := 'False'; ExternalWritable := 'False'} : Real;
      LowerSpeedLimit_Reached { ExternalAccessible := 'False'; ExternalVisible := 'False'; ExternalWritable := 'False'} : Bool;
      UpperSpeedLimit_Reached { ExternalAccessible := 'False'; ExternalVisible := 'False'; ExternalWritable := 'False'} : Bool;
      PowerTimer { ExternalAccessible := 'False'; ExternalVisible := 'False'; ExternalWritable := 'False'; S7_SetPoint := 'True'} : IEC_TIMER;
      HeatSinkTimer { ExternalAccessible := 'False'; ExternalVisible := 'False'; ExternalWritable := 'False'; S7_SetPoint := 'True'} : IEC_TIMER;
      HeatSourceTimer { ExternalAccessible := 'False'; ExternalVisible := 'False'; ExternalWritable := 'False'; S7_SetPoint := 'True'} : IEC_TIMER;
      VariableControlTimer { ExternalAccessible := 'False'; ExternalVisible := 'False'; ExternalWritable := 'False'; S7_SetPoint := 'True'} : IEC_TIMER;
      EngineRequired { ExternalAccessible := 'False'; ExternalVisible := 'False'; ExternalWritable := 'False'} : Bool := true;
      DT1_storage { ExternalAccessible := 'False'; ExternalVisible := 'False'; ExternalWritable := 'False'} : Real;
   END_VAR
   VAR_TEMP
      Dummy : Real;
      Target : Struct
         ID : Int;
         Error : Real;
         Target : Real;
         CurrentValue : Real;
         Kp : Real;
         Tn : Int;
         Tv : Int;
      END_STRUCT;
      T_Setpoint : Real;
      T_CurrentValue : Real;
      ManualControl_acv : Bool;
      DT_Source : Real;
      DT_Sink : Real;
      DT_VarCont : Real;
      ID : USInt;
      AddPressSafetyMargin : Real;
      ControlError : Real;
   END_VAR
   VAR CONSTANT
      KP_STEMP : Real := 20.0;
      TN_STEMP : Int := 120;
      i0 : Int := 0;
   END_VAR
BEGIN

REGION Network 1: Reset manual modes
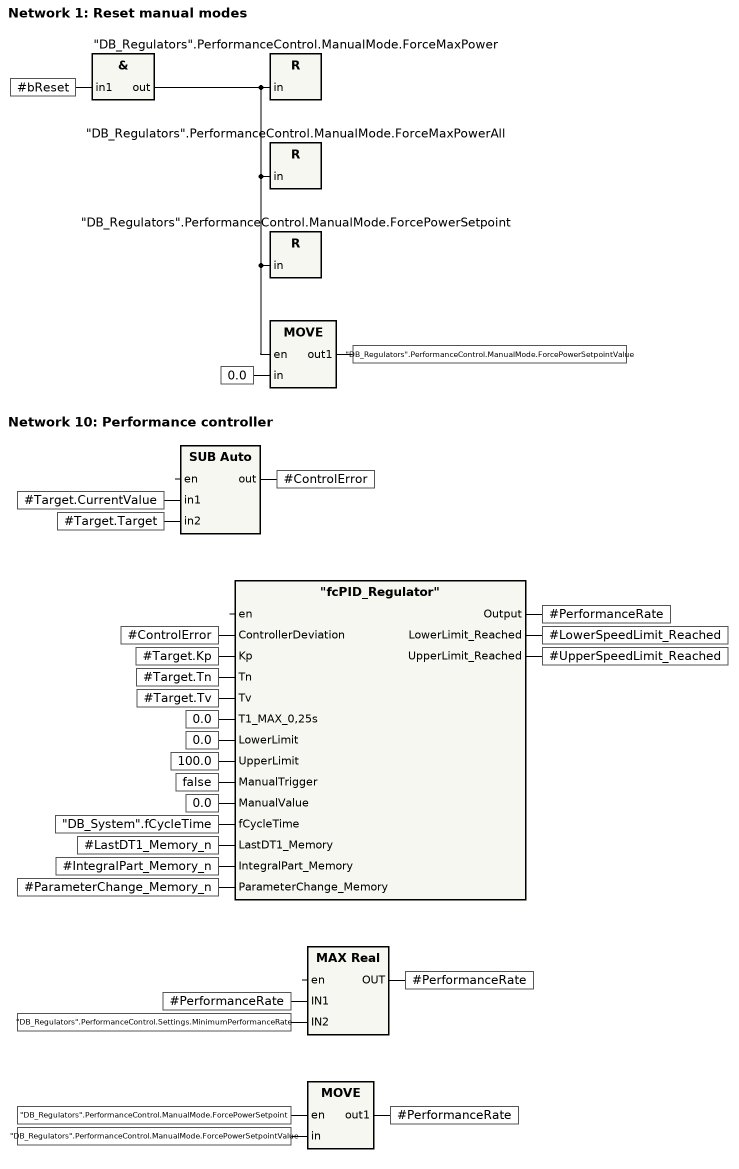
   IF #bReset THEN
       "DB_Regulators".PerformanceControl.ManualMode.ForceMaxPower := FALSE;
       "DB_Regulators".PerformanceControl.ManualMode.ForceMaxPowerAll := FALSE;
       "DB_Regulators".PerformanceControl.ManualMode.ForcePowerSetpoint := FALSE;
       "DB_Regulators".PerformanceControl.ManualMode.ForcePowerSetpointValue := 0.0;
   END_IF;
END_REGION

REGION Network 2 (SCL): Preset
   #ManualControl_acv := "DB_Regulators".PerformanceControl.ManualMode.ForceMaxPower OR "DB_Regulators".PerformanceControl.ManualMode.ForceMaxPowerAll OR "DB_Regulators".PerformanceControl.ManualMode.ForcePowerSetpoint;

   // Preset
   #Target.Tv := 0;
   #Target.Error := 20; // Positive value between 0.1-100, larger values mean the controller intervenes longer before the setpoint is reached, if it changes rapidly.
   #Target.Tn := REAL_TO_INT(#Target.Error * "DB_Regulators".PerformanceControl.Settings.Config.INCREASEWITHNORESTRICTION); // 
   #Target.Kp := 1;
END_REGION

REGION Network 3 (SCL): Heat sink control (Restrictions 1 & 2)
    IF "DB_Regulators".PerformanceControl.Settings.HeatSink.Control_Active THEN
      #T_Setpoint := "DB_Regulators".PerformanceControl.Settings.HeatSink.Setpoint;

       // NOTE! Feed Flow here means "discharge"
      IF "DB_Regulators".PerformanceControl.Settings.HeatSink.UseFeedFlow THEN
           // Heat sink discharge temperature
           #T_CurrentValue := "DB_AI".HBL_TT_518.Eng.fValue;
           #ID := USInt#2;
       ELSE
           // Heat sink suction temperature
           #T_CurrentValue := "DB_AI".HBL_TT_901.Eng.fValue;
           #ID := USInt#1;
       END_IF;
       #DT_Sink := #T_CurrentValue - #T_Setpoint;

       "Restriction"(ID := #ID,
                     Target := #T_Setpoint,
                     Value := #T_CurrentValue,
                     Kp := "DB_Regulators".PerformanceControl.Settings.HeatSink.Kp,
                     Tn := REAL_TO_INT("DB_Regulators".PerformanceControl.Settings.HeatSink.Tn),
                     Tv := #i0,
                     fCycleTime:= "DB_System".fCycleTime,
                     IO := #Target,
                     DT1_storage := #Dummy);
   END_IF;
END_REGION

REGION Network 4 (SCL): Heat source control (Restrictions 3 & 4)
    IF "DB_Regulators".PerformanceControl.Settings.HeatSource.Control_Active THEN
       #T_Setpoint := "DB_Regulators".PerformanceControl.Settings.HeatSource.Setpoint;

       // NOTE! "Feed flow" here means "suction"
       IF "DB_Regulators".PerformanceControl.Settings.HeatSource.UseFeedFlow THEN
           // Heat source suction temperature
           #T_CurrentValue := "DB_AI".HBL_TT_546.Eng.fValue;
           #ID := USInt#4;
       ELSE
           // Heat source discharge temperature
           #T_CurrentValue := "DB_AI".HBL_TT_542.Eng.fValue;
           #ID := USInt#3;

       END_IF;
       #DT_Source := #T_Setpoint - #T_CurrentValue;

       "Restriction"(ID := #ID,
                     Target := #T_Setpoint,
                     Value := #T_CurrentValue,
                     Kp := "DB_Regulators".PerformanceControl.Settings.HeatSource.Kp,
                     Tn := REAL_TO_INT("DB_Regulators".PerformanceControl.Settings.HeatSource.Tn),
                     Tv := #i0,
                     fCycleTime := "DB_System".fCycleTime,
                     IO := #Target,
                     DT1_storage := #Dummy);
   END_IF;
END_REGION

REGION Network 5 (SCL): Variable control (Restriction 6)
   IF "DB_Regulators".PerformanceControl.Settings.VariableControl.Control_Active AND "DB_Regulators".PerformanceControl.Settings.VariableControl.ReferenceID > 0 THEN
       #T_Setpoint := "DB_Regulators".PerformanceControl.Settings.VariableControl.Setpoint;

       CASE "DB_Regulators".PerformanceControl.Settings.VariableControl.ReferenceID OF
           1:
               #T_CurrentValue := "DB_AI".HBL_TT_901.Eng.fValue;
           2:
               #T_CurrentValue := "DB_AI".HBL_TT_518.Eng.fValue;
           3:
               #T_CurrentValue := "DB_Calc".HeatSink.DeltaT.fValue;
           4:
               #T_CurrentValue := "DB_AI".HBL_TT_542.Eng.fValue;
           5:
               #T_CurrentValue := "DB_AI".HBL_TT_546.Eng.fValue;
           6:
               #T_CurrentValue := "DB_Calc".HeatSource.DeltaT.fValue;
           7:
               #T_CurrentValue := 0; //Extern Temperature Sensor
           ELSE  // Statement section ELSE
               #T_CurrentValue := 0;
       END_CASE;
       #DT_VarCont := #T_CurrentValue - #T_Setpoint;

       "Restriction"(ID := 6,
                     Target := #T_Setpoint,
                     Value := #T_CurrentValue,
                     Kp := "DB_Regulators".PerformanceControl.Settings.VariableControl.Kp,
                     Tn := REAL_TO_INT("DB_Regulators".PerformanceControl.Settings.VariableControl.Tn),
                     Tv := #i0,
                     fCycleTime := "DB_System".fCycleTime,
                     IO := #Target,
                     DT1_storage := #Dummy);
   END_IF;
END_REGION

REGION Network 6 (SCL): Safety limit condensing pressure (Restriction 8)
   // If condensing temperature is close or above Heat sink feed temperature, increase safety margin  (-2K - 4K) difference   => (0 - 300kPa) extra
   #AddPressSafetyMargin := LIMIT_REAL(IN := ("DB_Calc".HighPressPart.CondenserSaturationTemperature.fValue - "DB_AI".HBL_TT_518.Eng.fValue + 2) * 50, MN := 0, MX := 300);

   // If condensing maximum pressure is close or above critical point, increase safety margin         (0 - 400kPa) difference => (0 - 200kPa) extra
   #AddPressSafetyMargin += LIMIT_REAL(IN := ("DB_CurrentSetting".System.Limits.p_CompressorOut_Max - "DB_CurrentSetting".Fluid.P_CriticalPoint) * 0.5, MN := 0, MX := 200);

   "Restriction"(ID:=8,
                 Target:="DB_CurrentSetting".System.Limits.p_CompressorOut_Max - 200.0 - #AddPressSafetyMargin,
                 Value:="DB_AI".HBL_PT_517.Eng.fValue,
                 Kp:=0.36,
                 Tn:=16,
                 Tv:=25,
                 fCycleTime := "DB_System".fCycleTime,
                 IO:=#Target,
                 DT1_storage:=#DT1_storage);
END_REGION

REGION Network 7 (SCL): Safety limit torque (Restriction 9)
   // ##REVIEW THIS!! Should be operating at 100% torque limit unless some good reason for it?
   // Safety limit compressor motor torque (110Nm @ 1500rpm)
   "Restriction"(ID:=9,
                 Target:=110.0*SQRT(1500/"DB_InverterDrives".HBL_SC_10.Stat.Speed.Eng.fValue),
                 Value:= "DB_InverterDrives".HBL_SC_10.Stat.Torque.Eng.fValue,
                 Kp:=0.04,
                 Tn:=3,
                 Tv:=#i0,
                 fCycleTime:= "DB_System".fCycleTime,
                 IO:=#Target,
                 DT1_storage:=#Dummy);
END_REGION

REGION Network 8 (SCL): Safety limit temperatures (Restriction 10, 11, 12, 14)
    // Safety limit compressor motor winding temperature
   "Restriction"(ID:=10,
                 Target:="DB_CurrentSetting".Compressor.Limits.T_Motor_Max - 5,
                 Value:="DB_AI".HBL_TT_20.Eng.fValue,
                 Kp:=#KP_STEMP,
                 Tn:=#TN_STEMP,
                 Tv:=#i0,
                 fCycleTime := "DB_System".fCycleTime,
                 IO:=#Target,
                 DT1_storage:=#Dummy);
   // Safety limit container air temperature
   "Restriction"(ID:=11,
                 Target:="DB_CurrentSetting".System.Limits.T_Housing_Max - 5,
                 Value:="DB_AI".HBL_TT_16.Eng.fValue,
                 Kp:=#KP_STEMP,
                 Tn:=#TN_STEMP,
                 Tv:=#i0,
                 fCycleTime := "DB_System".fCycleTime,
                 IO:=#Target,
                 DT1_storage:=#Dummy);
   // Safety limit control cabinet air temperature
   "Restriction"(ID:=12,
                 Target:="DB_CurrentSetting".StaticSetting.Limits.T_Cabinet_Max - 3,
                 Value:="DB_AI".HBL_TT_17.Eng.fValue,
                 Kp:=#KP_STEMP,
                 Tn:=#TN_STEMP,
                 Tv:=#i0,
                 fCycleTime := "DB_System".fCycleTime,
                 IO:=#Target,
                 DT1_storage:=#Dummy);
   // Safety limit compressor inverter temperature
   (*
   "Restriction"(ID:=13,
                 Target:="DB_CurrentSetting".CompressorTypes.Limits.T_Inverter_Max - 5,
                 Value:="DB_SensorInputs".Compressors.T19_Inverter,
                 Kp:=#KP_STEMP,
                 Tn:=#TN_STEMP,
                 Tv:=#i0,
                 fCycleTime:= "DB_System".fCycleTime,
                 IO:=#Target,
                 DT1_storage:=#Dummy);
   *)
   // Safety limit oil sump oil temperature (Max - 5°C)
   "Restriction"(ID:=14,
                 Target:="DB_CurrentSetting".Fluid.Limits.T_OilTemperature_Critical - 5,
                 Value:="DB_AI".HBL_TT_03.Eng.fValue,
                 Kp:=#KP_STEMP,
                 Tn:=#TN_STEMP,
                 Tv:=#i0,
                 fCycleTime := "DB_System".fCycleTime,
                 IO:=#Target,
                 DT1_storage:=#Dummy);
END_REGION

REGION Network 9 (SCL): Force max power
   // Bypass all power limitations. Self-protection limitations included
   IF "DB_Regulators".PerformanceControl.ManualMode.ForceMaxPowerAll THEN
       #Target.Error := 10.0;
       #Target.ID := 0;
       #Target.Kp  := #KP_STEMP;
       #Target.Tn  := #TN_STEMP;
   END_IF;
END_REGION

REGION Network 10: Performance controller
   // ###NOTSURE disable the manual mode (overwrites output instead in FB34)
   #ControlError := #Target.CurrentValue - #Target.Target;
   "fcPID_Regulator"(ControllerDeviation := #ControlError,
                     Kp := #Target.Kp,
                     Tn := #Target.Tn,
                     Tv := #Target.Tv,
                     "T1_MAX_0,25s" := 0.0,
                     LowerLimit := 0.0,
                     UpperLimit := 100.0,
                     ManualTrigger := false,
                     ManualValue := 0.0,
                     fCycleTime := "DB_System".fCycleTime,
                     LastDT1_Memory := #LastDT1_Memory_n,
                     IntegralPart_Memory := #IntegralPart_Memory_n,
                     ParameterChange_Memory := #ParameterChange_Memory_n,
                     Output => #PerformanceRate,
                     LowerLimit_Reached => #LowerSpeedLimit_Reached,
                     UpperLimit_Reached => #UpperSpeedLimit_Reached);
   #PerformanceRate := MAX(IN1 := #PerformanceRate, IN2 := "DB_Regulators".PerformanceControl.Settings.MinimumPerformanceRate);
   IF "DB_Regulators".PerformanceControl.ManualMode.ForcePowerSetpoint THEN
       #PerformanceRate := "DB_Regulators".PerformanceControl.ManualMode.ForcePowerSetpointValue;
   END_IF;
END_REGION

REGION Network 11 (SCL): Outputs
   //If there is no nagative restriction and the Powersetpoint is 100%. Don't show restrictions.
   IF #Target.Error > 0 AND #PerformanceRate >= 98 THEN 
       #Target.ID := 0;
   END_IF;

   // Local outputs
   IF #EngineRequired AND ("DB_State".State."5_Warmup" OR "DB_State".State."6_Running") THEN
       #Rate := #PerformanceRate;
   ELSE
       #Rate := 0;
   END_IF;

   "DB_Regulators".PerformanceControl.RestrictionID := #RestrictionID := #Target.ID;
   "DB_Regulators".PerformanceControl.TargetValue := #TargetValue := #Target.Target;
   "DB_Regulators".PerformanceControl.CurrentValue := #CurrentValue := #Target.CurrentValue;
   "DB_Regulators".PerformanceControl.fOut := #CompressorPerformanceSetpoint := #PerformanceRate;
END_REGION

REGION Network 12 (SCL): AdditionalSuperheatRequest
   // If the performance rate is below a minimum (X%) an additional superheat is required. The maximum required superheat (UpperAdditionalSuperheatLimit) is reached if the power requirement is 0;
   // Ab einer Leistung kleiner X% soll ein zusätzliches Superheat angefordert werden. Maximal MaximumAdditionalSuperheat
   #T_AddSuperheat_Controlled := MAX(IN1:= ("DB_Regulators".PerformanceControl.Settings.Config.MinimumPerformanceRequirement-#PerformanceRate)/"DB_Regulators".PerformanceControl.Settings.Config.MinimumPerformanceRequirement, 
                                     IN2:= 0)*"DB_Regulators".PerformanceControl.Settings.Config.MaximumAdditionalSuperheat;
END_REGION

REGION Network 13 (SCL): Validate standby/operational limits
   // Validate settings
   IF "DB_Regulators".PerformanceControl.Settings.HeatSink.DT_Limit_Standby < - "DB_Regulators".PerformanceControl.Settings.HeatSink.DT_Limit_Resume THEN
       "DB_Regulators".PerformanceControl.Settings.HeatSink.DT_Limit_Resume := "DB_Regulators".PerformanceControl.Settings.HeatSink.DT_Limit_Standby;
   END_IF;
   IF "DB_Regulators".PerformanceControl.Settings.HeatSource.DT_Limit_Standby < - "DB_Regulators".PerformanceControl.Settings.HeatSource.DT_Limit_Resume THEN
       "DB_Regulators".PerformanceControl.Settings.HeatSource.DT_Limit_Resume := "DB_Regulators".PerformanceControl.Settings.HeatSource.DT_Limit_Standby;
   END_IF;
   IF "DB_Regulators".PerformanceControl.Settings.VariableControl.DT_Limit_Standby < - "DB_Regulators".PerformanceControl.Settings.VariableControl.DT_Limit_Resume THEN
       "DB_Regulators".PerformanceControl.Settings.VariableControl.DT_Limit_Resume := "DB_Regulators".PerformanceControl.Settings.VariableControl.DT_Limit_Standby;
   END_IF;
END_REGION

REGION Network 14 (SCL): Running condition
   // 

   IF #EngineRequired THEN
       // Running condition is true, see if we need to reset it
       #PowerTimer.TON(IN:=("DB_Regulators".PerformanceControl.Settings.SwitchToStandby_timeDelay <> T#0s) AND 
                           (#PerformanceRate <= "DB_Regulators".PerformanceControl.Settings.MinimumPerformanceRate), PT := "DB_Regulators".PerformanceControl.Settings.SwitchToStandby_timeDelay + T#1ms);

       #HeatSinkTimer.TON(IN:= "DB_Regulators".PerformanceControl.Settings.HeatSink.Control_Active AND 
                               (#DT_Sink >= "DB_Regulators".PerformanceControl.Settings.HeatSink.DT_Limit_Standby), PT:= T#1s);
       #HeatSourceTimer.TON(IN:= "DB_Regulators".PerformanceControl.Settings.HeatSource.Control_Active AND 
                                (#DT_Source >= "DB_Regulators".PerformanceControl.Settings.HeatSource.DT_Limit_Standby), PT:= T#1s);
       #VariableControlTimer.TON(IN := "DB_Regulators".PerformanceControl.Settings.VariableControl.Control_Active AND 
                                       (#DT_VarCont >= "DB_Regulators".PerformanceControl.Settings.VariableControl.DT_Limit_Standby), PT := T#1s);
       IF (#PowerTimer.Q OR #HeatSinkTimer.Q OR #HeatSourceTimer.Q OR #VariableControlTimer.Q) AND NOT #ManualControl_acv THEN
           PRESET_TIMER("TIMER":=#PowerTimer,PT:=T#1ms);
           PRESET_TIMER("TIMER":=#HeatSinkTimer,PT:=T#1ms);    
           PRESET_TIMER("TIMER":=#HeatSourceTimer,PT:=T#1ms);
           PRESET_TIMER("TIMER" := #VariableControlTimer,PT := T#1ms);
           #EngineRequired := false;
       END_IF;
   ELSE
       // Running condition is false, see if we need to set it
       #PowerTimer.TOF(IN:=("DB_Regulators".PerformanceControl.Settings.SwitchToStandby_timeDelay <> T#0s) AND 
                           (#PerformanceRate <= "DB_Regulators".PerformanceControl.Settings.MinimumPerformanceRate), PT := "DB_Regulators".PerformanceControl.Settings.SwitchToStandby_timeDelay + T#1ms);
       #HeatSinkTimer.TOF(IN:="DB_Regulators".PerformanceControl.Settings.HeatSink.Control_Active AND 
                              (#DT_Sink > - "DB_Regulators".PerformanceControl.Settings.HeatSink.DT_Limit_Resume), PT:= T#1s);
       #HeatSourceTimer.TOF(IN:= "DB_Regulators".PerformanceControl.Settings.HeatSource.Control_Active AND 
                                 (#DT_Source > - "DB_Regulators".PerformanceControl.Settings.HeatSource.DT_Limit_Resume), PT:= T#1s);
       #VariableControlTimer.TOF(IN := "DB_Regulators".PerformanceControl.Settings.VariableControl.Control_Active AND 
                                       (#DT_VarCont > - "DB_Regulators".PerformanceControl.Settings.VariableControl.DT_Limit_Resume), PT := T#1s);
       IF NOT(#PowerTimer.Q OR #HeatSinkTimer.Q OR #HeatSourceTimer.Q OR #VariableControlTimer.Q) OR #ManualControl_acv THEN
           RESET_TIMER(#PowerTimer);
           RESET_TIMER(#HeatSinkTimer);
           RESET_TIMER(#HeatSourceTimer);
           RESET_TIMER(#VariableControlTimer);
           #EngineRequired := true;
       END_IF;
   END_IF;
   #RunningCondition:= #EngineRequired;
   "DB_Regulators".PerformanceControl.RunningCondition := #EngineRequired;
END_REGION
END_FUNCTION_BLOCK

FUNCTION "fcPID_Regulator" : Void   // FC54, FBD
{ S7_Optimized_Access := 'TRUE' }
VERSION : 0.1
// stored: AutoNumber true, IsIECCheckEnabled false, SetENOAutomatically false, UDAEnableTagReadback false
   VAR_INPUT
      ControllerDeviation : Real;
      Kp : Real;
      Tn : Real;
      Tv : Real;
      "T1_MAX_0,25s" : Real;
      LowerLimit : Real;
      UpperLimit : Real;
      ManualTrigger : Bool;
      ManualValue : Real;
      fCycleTime : Real;
   END_VAR
   VAR_OUTPUT
      Output : Real;
      LowerLimit_Reached : Bool;
      UpperLimit_Reached : Bool;
   END_VAR
   VAR_IN_OUT
      LastDT1_Memory : Real;
      IntegralPart_Memory : Real;
      ParameterChange_Memory : Real;
   END_VAR
   VAR_TEMP
      DifferentialFactor : Real;
      DT1 : Real;
      ProportionalPart : Real;
      "PI-Part" : Real;
      ResetFactor : Real;
   END_VAR
BEGIN

REGION Network 1 (SCL): Controller difference and calculation of proportional part
   #ProportionalPart := (#ControllerDeviation) * #Kp;
END_REGION

REGION Network 2 (SCL): DT1 formular
   #DT1 :=(#ControllerDeviation - #LastDT1_Memory) / (#"T1_MAX_0,25s" + #fCycleTime);

   //Stores Merk for the DT1 calculation of the next cycle
   #LastDT1_Memory += #DT1 * #fCycleTime;
END_REGION

REGION Network 3 (SCL): Calculation of the differential part factor
   // Reset Differential part if Tv=0 or ManaulValue active or DifferentialFactor=NAN or if Kp was changed
   IF #Tv = 0 OR #ManualTrigger OR "isNaN"(#DT1) THEN
       #DifferentialFactor := 0;
       #LastDT1_Memory := 0;
   ELSE
       #DifferentialFactor := #DT1 * #Kp * #Tv;
   END_IF;
END_REGION

REGION Network 4 (SCL): Calculation of the integral part
   // Reset Integal memory if Tn=0 or if IntegralPart_Memory=NaN
   IF (#Tn <> 0) AND "isNotNaN"(#IntegralPart_Memory) THEN
   //The integral part is calculated by the last integral part
       #IntegralPart_Memory +=           
       //plus the propotional part devided by the integral factor
       #ProportionalPart * (#fCycleTime / #Tn) -
       //in case of parameter changes on Kp an improving value must be substracted to balance the changes on Kp
       #ControllerDeviation * (#Kp - #ParameterChange_Memory);
   ELSE
       //Deactivates the integral part, if there's no valid number at Tn
       #IntegralPart_Memory := 0;
   END_IF;
END_REGION

REGION Network 5 (SCL): Combination of integral, proportional and differential parts and limit monitoring and switch to manual value
   #"PI-Part" := #ProportionalPart + #IntegralPart_Memory;

   IF #ManualTrigger THEN
       #Output := #ManualValue;
   ELSE
       //Limiting OutputValue to given limits
       #Output := LIMIT(MN := #LowerLimit, IN := #"PI-Part" + #DifferentialFactor, MX := #UpperLimit);
       //Show if a limit got reached
       #LowerLimit_Reached := NOT (#Output > #LowerLimit);
       #UpperLimit_Reached := #Output >= #UpperLimit;
   END_IF;
END_REGION

REGION Network 6 (SCL): Choice of feedback variable (wind up prevention) and calculation of the integral part
   #ResetFactor := (#fCycleTime / (#Tn+0.001)) * 3;// Factor between 1 and oo. 1 compensates Integral and stops sum to grow above maximum. Faktor 500 Sum is limited to match upper boundary after 1/20 Tn

   IF #ManualTrigger THEN
       //feeds back a manual-value-depending value, which is close to be constant and protects the controller against wind up
       #IntegralPart_Memory := #ManualValue - #ProportionalPart;
   ELSIF #"PI-Part" > #UpperLimit THEN
       //feeds back a upper-limit-depending value, which is close to be constant and protects the controller against wind up
       //#IntegralPart_Memory := #UpperLimit - #ProportionalPart;
       #IntegralPart_Memory += (#UpperLimit - #ProportionalPart) * #ResetFactor;
       #IntegralPart_Memory /= 1 + #ResetFactor;
   ELSIF #"PI-Part" < #LowerLimit THEN
       //feeds back a lower-limit-depending value, which is close to be constant and protects the controller against wind up
       //#IntegralPart_Memory := #LowerLimit - #ProportionalPart;
       #IntegralPart_Memory += (#LowerLimit - #ProportionalPart) * #ResetFactor;
       #IntegralPart_Memory /= 1 + #ResetFactor;
   END_IF;

   //If the Kp parameter is changing the integral part gets adjusted to it. Therefore the last Kp value must be stored for the next cycle
   #ParameterChange_Memory := #Kp;
END_REGION
END_FUNCTION

FUNCTION_BLOCK "SuperheatControl"   // FB23, FBD
TITLE = Pinch setpoint from superheat
{ S7_Optimized_Access := 'TRUE' }
VERSION : 0.1
// stored: AutoNumber true, IsIECCheckEnabled false, IsRetainMemResEnabled false, MemoryReserve 100, SetENOAutomatically false, UDAEnableTagReadback false
   VAR_INPUT
      bEnable { ExternalAccessible := 'False'; ExternalVisible := 'False'; ExternalWritable := 'False'} : Bool;   // 1 = enable controller 0 = disable controller
      bReset { ExternalAccessible := 'False'; ExternalVisible := 'False'; ExternalWritable := 'False'} : Bool;   // 1 = reset manual mode
      AdditionalSuperheat { ExternalAccessible := 'False'; ExternalVisible := 'False'; ExternalWritable := 'False'} : Real;
   END_VAR
   VAR_OUTPUT
      AddSuperheat { ExternalAccessible := 'False'; ExternalVisible := 'False'; ExternalWritable := 'False'} : Real;
   END_VAR
   VAR
      SuperheatSetpoint { ExternalAccessible := 'False'; ExternalVisible := 'False'; ExternalWritable := 'False'} : Real;
      PinchSetpoint { ExternalAccessible := 'False'; ExternalVisible := 'False'; ExternalWritable := 'False'} : Real;
      PinchPerformanceCurrent { ExternalAccessible := 'False'; ExternalVisible := 'False'; ExternalWritable := 'False'} : Real;
      Regulator { ExternalAccessible := 'False'; ExternalVisible := 'False'; ExternalWritable := 'False'} : Struct
         x_intern_1 { ExternalAccessible := 'False'; ExternalVisible := 'False'; ExternalWritable := 'False'} : Real;
         x_intern_2 { ExternalAccessible := 'False'; ExternalVisible := 'False'; ExternalWritable := 'False'} : Real;
         x_intern_3 { ExternalAccessible := 'False'; ExternalVisible := 'False'; ExternalWritable := 'False'} : Real;
      END_STRUCT;
      Enabled { ExternalAccessible := 'False'; ExternalVisible := 'False'; ExternalWritable := 'False'} : Bool;
      A3020 { ExternalAccessible := 'False'; ExternalVisible := 'False'; ExternalWritable := 'False'} : "fbHMIEvent";
   END_VAR
   VAR_TEMP
      PinchPerformance : Real;
      PIDControlInactive : Bool;   // Is true if pinch setpoint is externally controlled
   END_VAR
BEGIN

REGION Network 1: Reset manual mode
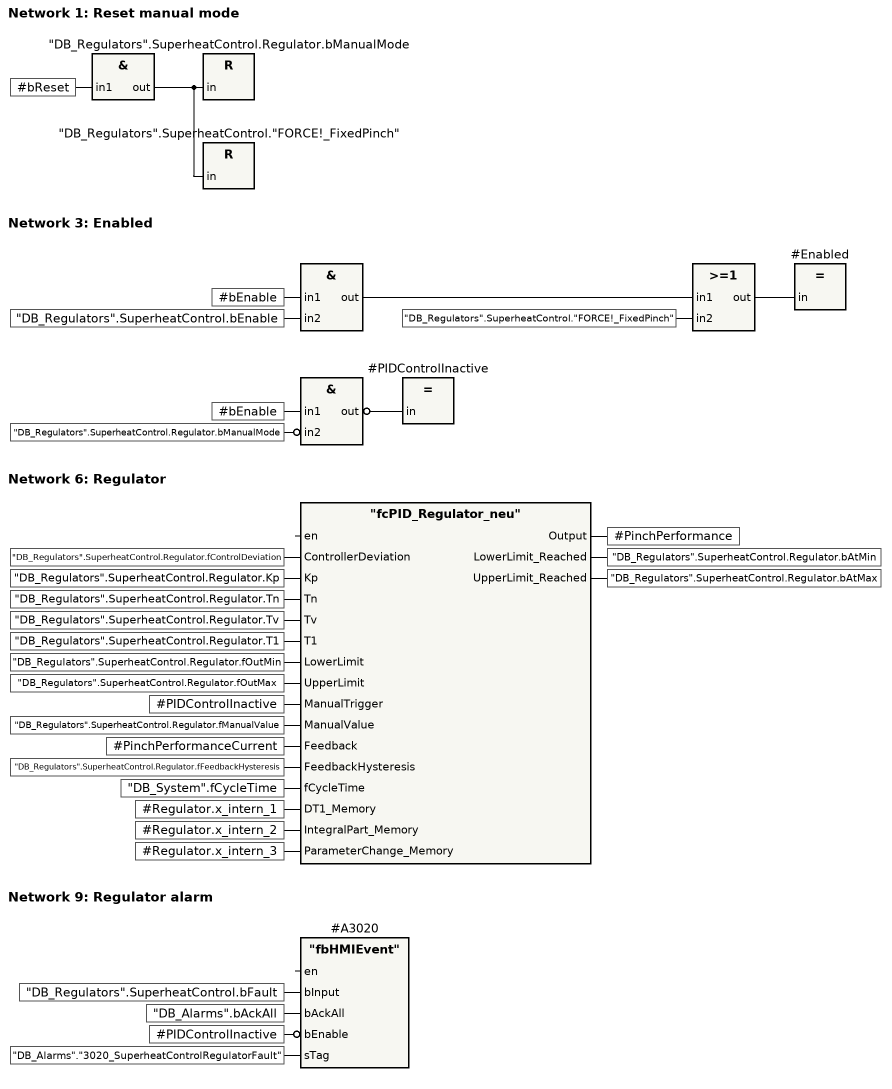
   IF #bReset THEN
       "DB_Regulators".SuperheatControl.Regulator.bManualMode := FALSE;
       "DB_Regulators".SuperheatControl."FORCE!_FixedPinch" := FALSE;
   END_IF;
END_REGION

REGION Network 2 (SCL): Manual values are given as Pinch, regulator works on "Pinch Performance"
   "DB_Regulators".SuperheatControl.Regulator.bManualMode := "DB_Regulators".SuperheatControl."FORCE!_FixedPinch";
END_REGION

REGION Network 3: Enabled
   // NOTE that we are not using the conventional bManual bit!!
   // Due to the difference between "Pinch Performance" and "Pinch"
   #Enabled := (#bEnable AND "DB_Regulators".SuperheatControl.bEnable) OR "DB_Regulators".SuperheatControl."FORCE!_FixedPinch";
   #PIDControlInactive := NOT (#bEnable AND NOT "DB_Regulators".SuperheatControl.Regulator.bManualMode);
END_REGION

REGION Network 4 (SCL): Superheat setpoint
   //Additional Superheat
   #AddSuperheat := #AdditionalSuperheat + "DB_Regulators".SuperheatControl.AdditionalSuperheat + "DB_CurrentSetting".Fluid.T_AdditionalSuperHeatEvaporator;

   #SuperheatSetpoint := 1.0 * "RecTarget"("DB_Regulators".SuperheatControl.fineTuningRecTarget) +
                         1.0 * #AddSuperheat;

   // Superheat setpoint
   IF "DB_State".State."6_Running" THEN
       #SuperheatSetpoint := #SuperheatSetpoint + 1.0 * "VapPerformance"(AddSuperheat := #AddSuperheat, Pinch := #PinchSetpoint);
   ELSE
       #SuperheatSetpoint := #SuperheatSetpoint + 0.5 * "VapPerformance"(AddSuperheat := #AddSuperheat, Pinch := #PinchSetpoint);

   END_IF;

   // Enforce a lower bound on the superheat
   #SuperheatSetpoint := MAX(IN1 := #SuperheatSetpoint, IN2 := "DB_CurrentSetting".System.Limits.T_SuperHeatCompressorIn_Min + 5.5);
END_REGION

REGION Network 5 (SCL): Deviation
   IF "DB_Regulators".SuperheatControl.Regulator.bManualMode = TRUE THEN
       "DB_Regulators".SuperheatControl.Regulator.fManualValue := LN(MAX(IN1 := "DB_Regulators".SuperheatControl."FORCE!_FixedPinch_Value", IN2 := 0.01)) * "DB_Regulators".SuperheatControl.ExponentialPinchFactor;
       "DB_Regulators".SuperheatControl.bFault := FALSE;
   ELSE
       //- Preset manual value to current pinch value to set controller to this value if inactive. Except if bManualMode whwre we directely set it to the target pinch performance
       //- Limited to 1K superhetat to prevent division by zero and critical low pinch values
       "DB_Regulators".SuperheatControl.Regulator.fManualValue := LN(MAX(IN1 := "DB_Calc".HeatSource.Pinch.fValue, IN2 := 1)) * "DB_Regulators".SuperheatControl.ExponentialPinchFactor;

       //Preset with current pinch as starting value if "FORCE!_FixedPinch is used
       "DB_Regulators".SuperheatControl."FORCE!_FixedPinch_Value" := "DB_Calc".HeatSource.Pinch.fValue;


       //Auto mode setpoint
       IF "isNaN"("DB_Calc".LowPressPart.CompressorSuperheat.fValue) OR "isNaN"(#SuperheatSetpoint) THEN
           "DB_Regulators".SuperheatControl.Regulator.fControlDeviation := 0;
           "DB_Regulators".SuperheatControl.bFault := TRUE;
       ELSE
           "DB_Regulators".SuperheatControl.Regulator.fControlDeviation := #SuperheatSetpoint - "DB_Calc".LowPressPart.CompressorSuperheat.fValue;
           "DB_Regulators".SuperheatControl.bFault := FALSE;
       END_IF;
   END_IF;

   //- Current pinch performance for informative reasons
   //- Limited to 0.1K to prevent division by zero 
   #PinchPerformanceCurrent := LN(MAX(IN1 := "DB_Calc".HeatSource.Pinch.fValue, IN2 := 0.1)) * "DB_Regulators".SuperheatControl.ExponentialPinchFactor;
END_REGION

REGION Network 6: Regulator
   "fcPID_Regulator_neu"(ControllerDeviation := "DB_Regulators".SuperheatControl.Regulator.fControlDeviation,
                         Kp := "DB_Regulators".SuperheatControl.Regulator.Kp,
                         Tn := "DB_Regulators".SuperheatControl.Regulator.Tn,
                         Tv := "DB_Regulators".SuperheatControl.Regulator.Tv,
                         T1 := "DB_Regulators".SuperheatControl.Regulator.T1,
                         LowerLimit := "DB_Regulators".SuperheatControl.Regulator.fOutMin,
                         UpperLimit := "DB_Regulators".SuperheatControl.Regulator.fOutMax,
                         ManualTrigger := #PIDControlInactive,
                         ManualValue := "DB_Regulators".SuperheatControl.Regulator.fManualValue,
                         Feedback := #PinchPerformanceCurrent,
                         FeedbackHysteresis := "DB_Regulators".SuperheatControl.Regulator.fFeedbackHysteresis,
                         fCycleTime := "DB_System".fCycleTime,
                         DT1_Memory := #Regulator.x_intern_1,
                         IntegralPart_Memory := #Regulator.x_intern_2,
                         ParameterChange_Memory := #Regulator.x_intern_3,
                         Output => #PinchPerformance,
                         LowerLimit_Reached => "DB_Regulators".SuperheatControl.Regulator.bAtMin,
                         UpperLimit_Reached => "DB_Regulators".SuperheatControl.Regulator.bAtMax);
END_REGION

REGION Network 7 (SCL): Convert Pinch Performance to Pinch
   //The PinchPerfomance value is interpreted logarithmically as pinch set point (-oo => 0K; 0 => 1K; 110 => 163K). 
   //Constant changes of PinchPerformance will cause only relative changes of the effective pinch. Pinch = e^(PinchPerformance/21,6)
   IF "DB_Regulators".SuperheatControl.Regulator.bManualMode = TRUE THEN
       "DB_Regulators".SuperheatControl.Regulator.fOut := "DB_Regulators".SuperheatControl."FORCE!_FixedPinch_Value";
   ELSE
       "DB_Regulators".SuperheatControl.Regulator.fOut := EXP(#PinchPerformance / "DB_Regulators".SuperheatControl.ExponentialPinchFactor);
       // Keep the manual value in sync to avoid discontinuities when switching from normal operation to Manual:
       //"DB_Regulators".SuperheatControl."FORCE!_FixedPinch_Value" := "DB_Regulators".SuperheatControl.Regulator.fOut;

   END_IF;
END_REGION

REGION Network 8 (SCL): Disable
   //IF #Enabled = FALSE THEN
   //    "DB_Regulators".SuperheatControl.Regulator.fOut := "DB_Regulators".SuperheatControl."FORCE!_FixedPinch_Value";
   //    "DB_Regulators".SuperheatControl.Regulator.bAtMin := FALSE;
   //    "DB_Regulators".SuperheatControl.Regulator.bAtMax := FALSE;
   //END_IF;
END_REGION

REGION Network 9: Regulator alarm
   #A3020(bInput := "DB_Regulators".SuperheatControl.bFault,   // "fbHMIEvent"
          bAckAll := "DB_Alarms".bAckAll,
          bEnable := NOT #PIDControlInactive,
          sTag := "DB_Alarms"."3020_SuperheatControlRegulatorFault");
END_REGION

REGION Network 10 (SCL): Mode
   // Only Auto or Manual in this regulator
   // Mode
   IF "DB_Regulators".SuperheatControl."FORCE!_FixedPinch" = TRUE THEN
       "DB_Regulators".SuperheatControl.nMode := 2;
   ELSE
       "DB_Regulators".SuperheatControl.nMode := 1;
   END_IF;
END_REGION
END_FUNCTION_BLOCK

FUNCTION "fcPID_Regulator_neu" : Void   // FC59, FBD
{ S7_Optimized_Access := 'TRUE' }
VERSION : 0.1
// stored: AutoNumber true, IsIECCheckEnabled false, SetENOAutomatically false, UDAEnableTagReadback false
   VAR_INPUT
      ControllerDeviation : Real;   // control deviation (to be eliminated by the PID control)
      Kp : Real;   // Proportional amplification factor (porportinal component / P)
      Tn : Real;   // Reset time (integral component / I)
      Tv : Real;   // Lead time (differential component / DT1)
      T1 : Real;   // Smoothing time constant (T1) of the differential part. PT1
      LowerLimit : Real;
      UpperLimit : Real;
      ManualTrigger : Bool;   // Set to Manual Value if active
      ManualValue : Real;
      Feedback : Real;   // Feeback of the manipulated variable (output). If they differ, the integral part is forced to correct this difference with Tn as correction time.
      FeedbackHysteresis : Real;   // The FeedbackHysteresics is an allowed error between feedback and output witch will be ignored
      fCycleTime : Real;
   END_VAR
   VAR_OUTPUT
      Output : Real;
      LowerLimit_Reached : Bool;
      UpperLimit_Reached : Bool;
   END_VAR
   VAR_IN_OUT
      DT1_Memory : Real;
      IntegralPart_Memory : Real;
      ParameterChange_Memory : Real;
   END_VAR
   VAR_TEMP
      DifferentialFactor : Real;
      DT1 : Real;
      ProportionalPart : Real;
      "PI-Part" : Real;
      ResetFactor : Real;
   END_VAR
BEGIN

REGION Network 1 (SCL): Controller difference and calculation of proportional part
   #ProportionalPart := (#ControllerDeviation) * #Kp;
END_REGION

REGION Network 2 (SCL): DT1 simulation formular
   // NOTE: can be replaced with an instance of FC58 DT1, if this becomes an FB
   #DT1 := (#ControllerDeviation - #DT1_Memory) / (#T1 + #fCycleTime);

   //Stores Merk for the DT1 calculation of the next cycle
   #DT1_Memory += #DT1 * #fCycleTime;
END_REGION

REGION Network 3 (SCL): Calculation of the differential part factor
   // Reset Differential part if Tv=0 or ManaulValue active or DifferentialFactor=NAN or if Kp was changed
   IF #Tv = 0 OR #ManualTrigger OR "isNaN"(#DT1) THEN
       #DifferentialFactor := 0;
       #DT1_Memory := 0;
   ELSE
       #DifferentialFactor := #DT1 * #Kp * #Tv;
   END_IF;
END_REGION

REGION Network 4 (SCL): Calculation of the integral part
   // Reset Integal memory if Tn=0 or if IntegralPart_Memory=NaN
   IF (#Tn <> 0) AND "isNotNaN"(#IntegralPart_Memory) THEN
       //The integral part is calculated by the last integral part
       #IntegralPart_Memory +=
       //plus the propotional part devided by the integral factor
       #ProportionalPart * (#fCycleTime / #Tn) -
       //in case of parameter changes on Kp an improving value must be substracted to balance the changes on Kp
       #ControllerDeviation * (#Kp - #ParameterChange_Memory);
   ELSE
       //Deactivates the integral part, if there's no valid number at Tn
       #IntegralPart_Memory := 0;
   END_IF;
END_REGION

REGION Network 5 (SCL): Combination of integral, proportional and differential parts and limit monitoring and switch to manual value
   #"PI-Part" := #ProportionalPart + #IntegralPart_Memory;

   IF #ManualTrigger THEN
       #Output := #ManualValue;
   ELSE
       //Limiting OutputValue to given limits
       #Output := LIMIT(MN := #LowerLimit, IN := #"PI-Part" + #DifferentialFactor, MX := #UpperLimit);
       //Show if a limit got reached
       #LowerLimit_Reached := #Output <= #LowerLimit;
       #UpperLimit_Reached := #Output >= #UpperLimit;
   END_IF;
END_REGION

REGION Network 6 (SCL): Choice of feedback variable (wind up prevention) and calculation of the integral part
   #ResetFactor := (#fCycleTime / (#Tn + 0.001)) * 3;// Factor between 1 and oo. 1 compensates Integral and stops sum to grow above maximum. Faktor 500 Sum is limited to match upper boundary after 1/20 Tn


   IF #ManualTrigger THEN
       //feeds back a manual-value-depending value, which is close to be constant and protects the controller against wind up
       #IntegralPart_Memory := #ManualValue - #ProportionalPart;
   ELSIF #"PI-Part" > #UpperLimit THEN
       //feeds back a upper-limit-depending value, which is close to be constant and protects the controller against wind up
       //#IntegralPart_Memory := #UpperLimit - #ProportionalPart;
       #IntegralPart_Memory += (#UpperLimit - #ProportionalPart) * #ResetFactor;
       #IntegralPart_Memory /= 1 + #ResetFactor;
   ELSIF #"PI-Part" < #LowerLimit THEN
       //feeds back a lower-limit-depending value, which is close to be constant and protects the controller against wind up
       //#IntegralPart_Memory := #LowerLimit - #ProportionalPart;
       #IntegralPart_Memory += (#LowerLimit - #ProportionalPart) * #ResetFactor;
       #IntegralPart_Memory /= 1 + #ResetFactor;
   ELSIF #"PI-Part" > #Feedback + #FeedbackHysteresis THEN
       #IntegralPart_Memory += ((#Feedback + #FeedbackHysteresis) - #ProportionalPart) * #ResetFactor / 3;
       #IntegralPart_Memory /= 1 + #ResetFactor / 3;
   ELSIF #"PI-Part" < #Feedback - #FeedbackHysteresis THEN
       #IntegralPart_Memory += ((#Feedback - #FeedbackHysteresis) - #ProportionalPart) * #ResetFactor / 3;
       #IntegralPart_Memory /= 1 + #ResetFactor / 3;
   END_IF;

   //If the Kp parameter is changing the integral part gets adjusted to it. Therefore the last Kp value must be stored for the next cycle
   #ParameterChange_Memory := #Kp;
END_REGION
END_FUNCTION

FUNCTION_BLOCK "PinchControl"   // FB44, FBD
TITLE = Pinch setpoint to expansion valve position
{ S7_Optimized_Access := 'TRUE' }
VERSION : 0.1
// stored: AutoNumber true, IsIECCheckEnabled false, IsRetainMemResEnabled false, MemoryReserve 40, SetENOAutomatically false, UDAEnableTagReadback false
   VAR_INPUT
      bEnable { ExternalAccessible := 'False'; ExternalVisible := 'False'; ExternalWritable := 'False'} : Bool;   // 1 = enable controller, 0 = disable controller
      bReset { ExternalAccessible := 'False'; ExternalVisible := 'False'; ExternalWritable := 'False'} : Bool;
      AddSuperheat { ExternalAccessible := 'False'; ExternalVisible := 'False'; ExternalWritable := 'False'} : Real;
   END_VAR
   VAR_OUTPUT
      EvaporationPressureLimitation { ExternalAccessible := 'False'; ExternalVisible := 'False'; ExternalWritable := 'False'} : Bool;
      CurrentPressureTarged { ExternalAccessible := 'False'; ExternalVisible := 'False'; ExternalWritable := 'False'} : Real;
   END_VAR
   VAR
      Regulator { ExternalAccessible := 'False'; ExternalVisible := 'False'; ExternalWritable := 'False'} : Struct
         x_intern_1 { ExternalAccessible := 'False'; ExternalVisible := 'False'; ExternalWritable := 'False'} : Real;
         x_intern_2 { ExternalAccessible := 'False'; ExternalVisible := 'False'; ExternalWritable := 'False'} : Real;
         x_intern_3 { ExternalAccessible := 'False'; ExternalVisible := 'False'; ExternalWritable := 'False'} : Real;
      END_STRUCT;
      AddPinch_RateOfSourceChange { ExternalAccessible := 'False'; ExternalVisible := 'False'; ExternalWritable := 'False'} : Real;
      Enabled { ExternalAccessible := 'False'; ExternalVisible := 'False'; ExternalWritable := 'False'} : Bool;
      A3030 { ExternalAccessible := 'False'; ExternalVisible := 'False'; ExternalWritable := 'False'} : "fbHMIEvent";
   END_VAR
   VAR_TEMP
      PIDControlInactive : Bool;   // if true set "#StaticOutputValue" to expansionvalves
      StaticOutputValue : Real;   // setpoint for expansionfalves if not "PIDControlInactive"
   END_VAR
   VAR CONSTANT
      EXP_VLV_PID_CALMING : Real := 27.0;   // Super Heat Temperature that reduces Control Ampfication by 64%
   END_VAR
BEGIN

REGION Network 1: Reset manual mode
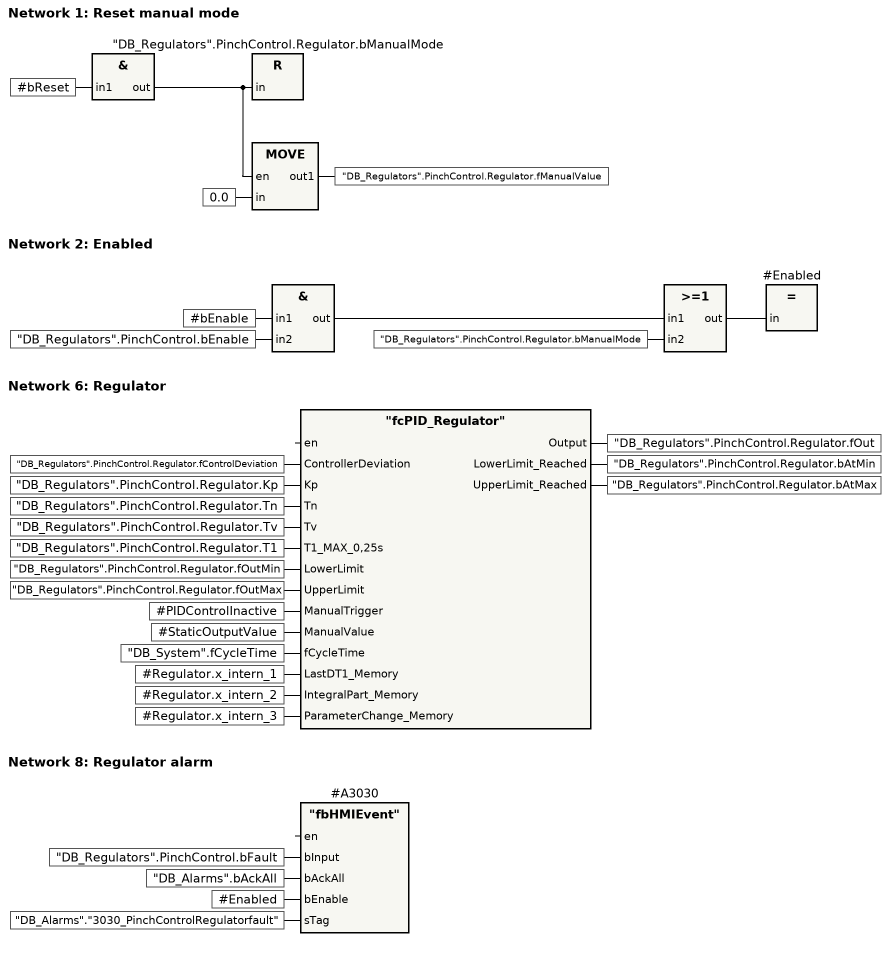
   IF #bReset THEN
       "DB_Regulators".PinchControl.Regulator.bManualMode := FALSE;
       "DB_Regulators".PinchControl.Regulator.fManualValue := 0.0;
   END_IF;
END_REGION

REGION Network 2: Enabled
   #Enabled := (#bEnable AND "DB_Regulators".PinchControl.bEnable) OR "DB_Regulators".PinchControl.Regulator.bManualMode;
END_REGION

REGION Network 3 (SCL): Static output
   // ###CHANGE: Added complete network:
   // If the controller is inactive and the expansion valve and the controller is set to an fixed value.
   IF ("DB_Regulators".PinchControl.Regulator.bManualMode) THEN
       // Set expansion valve to manual setpoint
       #StaticOutputValue := "DB_Regulators".PinchControl.Regulator.fManualValue;
   ELSIF ("DB_State".State."4_Start") THEN
       //Set expansion valves to fixed opening on startup
       //###CHANGE: The function to close the expansion valve if the compressor is stopped in dryout.
       //###CHANGE: Added the flag "DB_Regulators".PurgeControl.bDone = 0 since in state 4, in dyout (after purge), the "DB_Regulators".PurgeControl.bSpinning is zero but the comperssor is turning again. 
       IF ("DB_Regulators".PurgeControl.bSpinning = 0 AND "DB_Regulators".PurgeControl.bDone = 0) THEN
           #StaticOutputValue := 0;
       //###CHANGE: New function TO limit massflow on dryout with already filled evaporator at evaporation pressure > 300kPa.    
       ELSIF ("DB_AI".HBL_PT_572.Eng.fValue > 300.0) THEN   // 300kPa is larger than dryout pressure and sat at ~minimalinlet temperature. // 300kPa should be auto calculated or part of the dataset
           //###Note: With more than 300kPa we can assume that the evaporator is still filled and an additional amount of refrigerant would not be helpful
           #StaticOutputValue := "DB_CurrentSetting".MissingSetting.System.ExpansionValvePositionStartCold;
       ELSE
           #StaticOutputValue := "DB_CurrentSetting".MissingSetting.System.ExpansionValvePositionStart;
       END_IF;
   ELSIF (NOT #Enabled) THEN
       // Close expansion valve if inactive
       #StaticOutputValue := 0;
   END_IF;

   //Inactivate PID controler if a upper condition is fulfilled. Controler is reset to current output if true
   #PIDControlInactive := NOT #Enabled OR "DB_State".State."4_Start"OR"DB_Regulators".PinchControl.Regulator.bManualMode;
END_REGION

REGION Network 4 (SCL): Pinch setpoint
   // Setpoint is the pinch from the superheat regulator
   "DB_Regulators".PinchControl.fSetpoint := "DB_Regulators".SuperheatControl.Regulator.fOut;

   // Additional superheat
   "DB_Regulators".PinchControl.fSetpoint += 0.35 * #AddSuperheat * LIMIT_REAL(IN := "DB_Regulators".PinchControl.fSetpoint /"DB_Calc".LowPressPart.CompressorSuperheat.fValue, MN := 0,MX:=1); // Pilot-control-filter to bypass additional superheat to the pinch controller

   // Preliminary setpoint modification to counteract source temperature changes
   #AddPinch_RateOfSourceChange := -3.0 * "DB_Calc".HeatSource.TemperatureRateOfChange.fValue;

   IF #AddPinch_RateOfSourceChange > -0.75 * "DB_Regulators".PinchControl.fSetpoint THEN //Maximum compensation is 75% of unmodified Setpoint
       "DB_Regulators".PinchControl.fSetpoint += #AddPinch_RateOfSourceChange;
   ELSE
       //The internal value of the DT1-Block is also corrected by the leftover to enable a rapid response in case of a change of direction.
       (*#DT1_Merker_intern -= #AddPinch_RateOfSourceChange + 0.75 * #DB_Regulators.ExpansionValve.fSetpoint;*)
       //To avoid overcorrection the temperature change correction is limited to the left 25%.
       "DB_Regulators".PinchControl.fSetpoint *= 0.25;
   END_IF;
END_REGION

REGION Network 5 (SCL): Deviation
   //The control error is the difference between current pinch value and pinch setpoint.
   IF ("DB_Calc".HeatSource.Pinch.bError = TRUE) OR "isNaN"("DB_Regulators".PinchControl.fSetpoint) OR ("DB_Calc".Misc.EvaporatorDischargePressureMean.bError = TRUE) THEN
       "DB_Regulators".PinchControl.Regulator.fControlDeviation := 0;
       "DB_Regulators".PinchControl.bFault := TRUE;
   ELSE
       "DB_Regulators".PinchControl.bFault := FALSE;
       "DB_Regulators".PinchControl.Regulator.fControlDeviation := "DB_Calc".HeatSource.Pinch.fValue - "DB_Regulators".PinchControl.fSetpoint;

       // Maximum suction pressure protection
       // The target evaporation temperature should ensure a boiling pressure of no more than 1000 kPa (Maximum Limit - 100kPa). For this purpose, the control error is limited in case of a high evaporation pressure/temperature.
       IF "DB_Regulators".PinchControl.Regulator.fControlDeviation > (("DB_CurrentSetting".Compressor.Limits.p_CrankCase_Max - 100.0) - "DB_Calc".Misc.EvaporatorDischargePressureMean.fValue) THEN
           "DB_Regulators".PinchControl.Regulator.fControlDeviation := (("DB_CurrentSetting".Compressor.Limits.p_CrankCase_Max - 100.0) - "DB_Calc".Misc.EvaporatorDischargePressureMean.fValue) / 10.0;
           #EvaporationPressureLimitation := True;
       ELSE
           #EvaporationPressureLimitation := False;
       END_IF;

       // Current pressure target for visualisation and debugging
       #CurrentPressureTarged := "DB_Regulators".PinchControl.Regulator.fControlDeviation + "DB_Calc".Misc.EvaporatorDischargePressureMean.fValue;

       //Adapt Pinch control Kp-factor:
       //We need this function because an unloaded ("empty") evaporator reacts very sensitively to a changed refrigerant quantity. Empty or unloaded always means relatively much superheat, so that we can fine-tune it with this value.
       //The Kp factor depends on the Superheat after the Evaporator. If there is much superheat, the kp is smaller and if the superheat gets to zero it gets closer to the preset factor (3.0). A superheat of #EXP_VLV_PID_CALMING (14K) reduces Kp by 64% and a superheat of 2*#EXP_VLV_PID_CALMING reduces the Kp by 86%.
       "DB_Regulators".PinchControl.Regulator.Kp := 0.8 * LIMIT_REAL(IN := EXP((0.5 * "DB_Regulators".PinchControl.Regulator.fControlDeviation - "DB_Calc".LowPressPart.EvaporatorSuperheat.fValue) / #EXP_VLV_PID_CALMING), MN := 0.1, MX := 1);

       // The Lower limit for the expansion valve position can be increased on warmup
       // To ensure a minimal "heat" flow a minimal leakage might be helpful 
       IF "DB_State".State."5_Warmup" THEN
           "DB_Regulators".PinchControl.Regulator.fOutMin := "DB_CurrentSetting".MissingSetting.System.ExpansionValvePositionStart;
       ELSE
           "DB_Regulators".PinchControl.Regulator.fOutMin := 2.5;
       END_IF;
   END_IF;
END_REGION

REGION Network 6: Regulator
   "fcPID_Regulator"(ControllerDeviation := "DB_Regulators".PinchControl.Regulator.fControlDeviation,
                     Kp := "DB_Regulators".PinchControl.Regulator.Kp,
                     Tn := "DB_Regulators".PinchControl.Regulator.Tn,
                     Tv := "DB_Regulators".PinchControl.Regulator.Tv,
                     "T1_MAX_0,25s" := "DB_Regulators".PinchControl.Regulator.T1,
                     LowerLimit := "DB_Regulators".PinchControl.Regulator.fOutMin,
                     UpperLimit := "DB_Regulators".PinchControl.Regulator.fOutMax,
                     ManualTrigger := #PIDControlInactive,
                     ManualValue := #StaticOutputValue,
                     fCycleTime := "DB_System".fCycleTime,
                     LastDT1_Memory := #Regulator.x_intern_1,
                     IntegralPart_Memory := #Regulator.x_intern_2,
                     ParameterChange_Memory := #Regulator.x_intern_3,
                     Output => "DB_Regulators".PinchControl.Regulator.fOut,
                     LowerLimit_Reached => "DB_Regulators".PinchControl.Regulator.bAtMin,
                     UpperLimit_Reached => "DB_Regulators".PinchControl.Regulator.bAtMax);
END_REGION

REGION Network 7 (SCL): Disable
   IF #PIDControlInactive = True THEN
       "DB_Regulators".PinchControl.Regulator.fOut := #StaticOutputValue;
       "DB_Regulators".PinchControl.Regulator.bAtMin := FALSE;
       "DB_Regulators".PinchControl.Regulator.bAtMax := FALSE;
   END_IF;
END_REGION

REGION Network 8: Regulator alarm
   #A3030(bInput := "DB_Regulators".PinchControl.bFault,   // "fbHMIEvent"
          bAckAll := "DB_Alarms".bAckAll,
          bEnable := #Enabled,
          sTag := "DB_Alarms"."3030_PinchControlRegulatorfault");
END_REGION

REGION Network 9 (SCL): Mode
   // Mode
   IF "DB_Regulators".PinchControl.Regulator.bManualMode = TRUE THEN
       "DB_Regulators".PinchControl.nMode := 2;
   ELSIF "DB_Regulators".PinchControl.bEnable = TRUE THEN
       "DB_Regulators".PinchControl.nMode := 1;
   ELSE
       "DB_Regulators".PinchControl.nMode := 0;
   END_IF;
END_REGION
END_FUNCTION_BLOCK

FUNCTION_BLOCK "fbTemperatureController2"
TITLE = Heating and cooling control
{ S7_Optimized_Access := 'TRUE' }
VERSION : 0.1
//2-sided on/off control
   VAR_INPUT 
      sTemperature : "stCalcValue";   // Process value
      bEnable : Bool;
      bReset : Bool;   // 1 = reset manual modes
   END_VAR

   VAR_OUTPUT 
      bHeating : Bool;
      bCooling : Bool;
      bAtSetpoint : Bool;
   END_VAR

   VAR_IN_OUT 
      sTag : "stTemperatureController2";
   END_VAR

   VAR 
      Heating { S7_SetPoint := 'False'} : "fbHysteresis";
      Cooling : "fbHysteresis";
      Enabled { S7_SetPoint := 'True'} : Bool;
   END_VAR

   VAR_TEMP 
      fHeatingSetpoint : Real;
      fCoolingSetpoint : Real;
   END_VAR


BEGIN
	// 2-sided on/off temperature controller
	// Active heating & active cooling
	// Variant of fbOnOffController but with two regulation thresholds
	
	// Reset manual modes.
	IF #bReset THEN
	    #sTag.bManualMode := FALSE;
	    #sTag.fManualCoolingSetpoint := 0.0;
	    #sTag.fManualHeatingSetpoint := 0.0;
	    #sTag.bManualOverride := FALSE;
	    #sTag.nOverrideState := 0;
	END_IF;
	
	IF #sTag.bManualOverride = TRUE THEN
	    // In manual override, everything is awesome
	    #sTag.bAtSetpoint := TRUE;
	    #sTag.bFault := FALSE;
	    CASE #sTag.nOverrideState OF
	        0: // Off
	            #sTag.bHeating := FALSE;
	            #sTag.bCooling := FALSE;
	        1: // Heating
	            #sTag.bHeating := TRUE;
	            #sTag.bCooling := FALSE;
	        2: // Cooling
	            #sTag.bHeating := FALSE;
	            #sTag.bCooling := TRUE;
	    END_CASE;
	ELSE
	    // Choose setpoint
	    IF #sTag.bManualMode = TRUE THEN
	        #fHeatingSetpoint := #sTag.fManualHeatingSetpoint;
	        #fCoolingSetpoint := #sTag.fManualCoolingSetpoint;
	    ELSE
	        #fHeatingSetpoint := #sTag.fHeatingSetpoint;
	        #fCoolingSetpoint := #sTag.fCoolingSetpoint;
	    END_IF;
	
	    // Enabled when enabled from process and from HMI (Auto), or in Manual mode
	    #Enabled := (#bEnable AND #sTag.bEnable) OR #sTag.bManualMode;
	
	    // Run controller
	    IF #Enabled = TRUE AND #sTemperature.bError = FALSE AND (#fHeatingSetpoint < #fCoolingSetpoint) THEN
	        #Heating(fValue := #sTemperature.fValue, fLimit := #fHeatingSetpoint, fHysteresis := 0.5, bType := 0, bOutput => #sTag.bHeating);
	        #Cooling(fValue := #sTemperature.fValue, fLimit := #fCoolingSetpoint, fHysteresis := 0.5, bType := 1, bOutput => #sTag.bCooling);
	        #sTag.bAtSetpoint := NOT(#sTag.bHeating) AND NOT(#sTag.bCooling);
	    ELSE
	        #sTag.bAtSetpoint := FALSE;
	        #sTag.bHeating := FALSE;
	        #sTag.bCooling := FALSE;
	    END_IF;
	
	    // Controller fault
	    #sTag.bFault := #sTemperature.bError;
	    
	END_IF;
	
	// Mode
	IF #sTag.bManualOverride = TRUE THEN
	    #sTag.nMode := 3;
	ELSIF #sTag.bManualMode = TRUE THEN
	    #sTag.nMode := 2;
	ELSIF #sTag.bEnable = TRUE THEN
	    #sTag.nMode := 1;
	ELSE
	    #sTag.nMode := 0;
	END_IF;
	
	// Local outputs
	#bHeating := #sTag.bHeating;
	#bCooling := #sTag.bCooling;
	#bAtSetpoint := #sTag.bAtSetpoint;
	
END_FUNCTION_BLOCK

FUNCTION_BLOCK "OilHeating"   // FB17, FBD
TITLE = Crankcase oil sump heating control
{ S7_Optimized_Access := 'TRUE' }
VERSION : 0.1
// stored: AutoNumber true, IsIECCheckEnabled false, IsRetainMemResEnabled false, MemoryReserve 100, SetENOAutomatically false, UDAEnableTagReadback false
   VAR_INPUT
      bEnable { ExternalAccessible := 'False'; ExternalVisible := 'False'; ExternalWritable := 'False'} : Bool;
      bReset { ExternalAccessible := 'False'; ExternalVisible := 'False'; ExternalWritable := 'False'} : Bool;   // 1 = reset manual modes
   END_VAR
   VAR
      sHeaterControl { ExternalAccessible := 'False'; ExternalVisible := 'False'; ExternalWritable := 'False'} : "fbOnOffRegulator";
      bHeating { ExternalAccessible := 'False'; ExternalVisible := 'False'; ExternalWritable := 'False'; S7_SetPoint := 'True'} : Bool;
      A5000 { ExternalAccessible := 'False'; ExternalVisible := 'False'; ExternalWritable := 'False'; S7_SetPoint := 'True'} : "fbDigitalAlarm";
      A5001 { ExternalAccessible := 'False'; ExternalVisible := 'False'; ExternalWritable := 'False'; S7_SetPoint := 'True'} : "fbDigitalAlarm";
   END_VAR
   VAR_TEMP
      fSetpoint : Real;
   END_VAR
BEGIN

REGION Network 1 (SCL): Setpoint selection
   // Heating setpoint selection
   #fSetpoint := MAX(IN1 := "DB_CurrentSetting".VariableSetting.OilHeatSetpoint_min, IN2 := "DB_Calc".Compressor.CrankcaseSaturationTemperature.fValue + "DB_Regulators".OilHeating.fOilSuperheat);
   // Heating setpoint limitation
   "DB_Regulators".OilHeating.Controller.fSetpoint := MIN(IN1:= #fSetpoint, IN2:= "DB_CurrentSetting".Fluid.Limits.T_OilTemperature_Critical - 15);
END_REGION

REGION Network 2: Regulator
   // Additional criteria for running: crankcase wall temperatures are not above limit
   // Use the alarms to set time delay & hysteresis to prevent frequent triggering
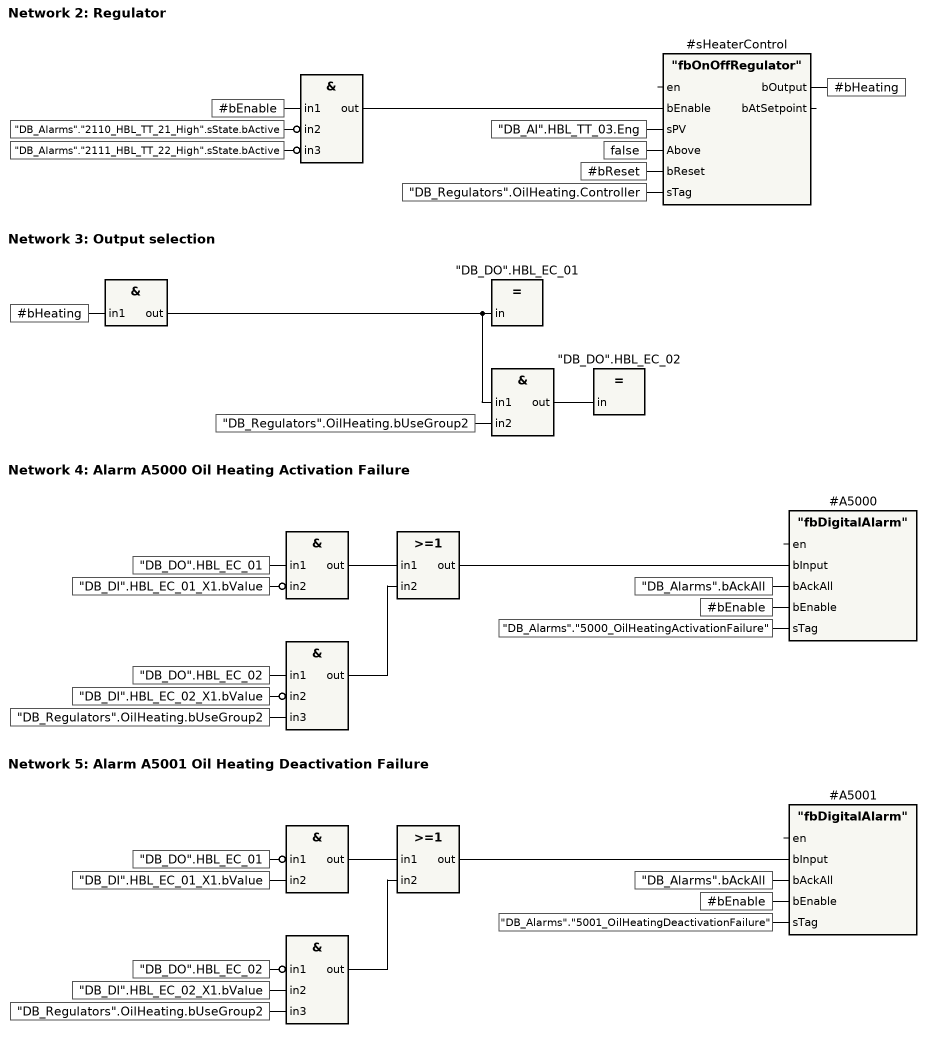
   #sHeaterControl(bEnable := #bEnable AND NOT "DB_Alarms"."2110_HBL_TT_21_High".sState.bActive AND NOT "DB_Alarms"."2111_HBL_TT_22_High".sState.bActive,   // "fbOnOffRegulator"
                   sPV := "DB_AI".HBL_TT_03.Eng,
                   Above := false,
                   bReset := #bReset,
                   sTag := "DB_Regulators".OilHeating.Controller,
                   bOutput => #bHeating);
END_REGION

REGION Network 3: Output selection
   // Selection of heater groups is manual for now. If programmatic selection is needed, change the code here :-)
   "DB_DO".HBL_EC_01 := #bHeating;
   "DB_DO".HBL_EC_02 := #bHeating AND "DB_Regulators".OilHeating.bUseGroup2;
END_REGION

REGION Network 4: Alarm A5000 Oil Heating Activation Failure
   #A5000(bInput := ("DB_DO".HBL_EC_01 AND NOT "DB_DI".HBL_EC_01_X1.bValue) OR ("DB_DO".HBL_EC_02 AND NOT "DB_DI".HBL_EC_02_X1.bValue AND "DB_Regulators".OilHeating.bUseGroup2),   // "fbDigitalAlarm"
          bAckAll := "DB_Alarms".bAckAll,
          bEnable := #bEnable,
          sTag := "DB_Alarms"."5000_OilHeatingActivationFailure");
END_REGION

REGION Network 5: Alarm A5001 Oil Heating Deactivation Failure
   #A5001(bInput := (NOT "DB_DO".HBL_EC_01 AND "DB_DI".HBL_EC_01_X1.bValue) OR (NOT "DB_DO".HBL_EC_02 AND "DB_DI".HBL_EC_02_X1.bValue AND "DB_Regulators".OilHeating.bUseGroup2),   // "fbDigitalAlarm"
          bAckAll := "DB_Alarms".bAckAll,
          bEnable := #bEnable,
          sTag := "DB_Alarms"."5001_OilHeatingDeactivationFailure");
END_REGION
END_FUNCTION_BLOCK

FUNCTION_BLOCK "fbOnOffRegulator"
{ S7_Optimized_Access := 'TRUE' }
VERSION : 0.1
   VAR_INPUT 
      bEnable : Bool;   // Enable from process. 1 = enabled, 0 = disabled
      sPV : "stCalcValue";   // Process value
      Above : Bool;   // 1 = regulate when above threshold, 0 = regulate when below threshold
      bReset : Bool;   // 1 = reset manual modes
   END_VAR

   VAR_OUTPUT 
      bOutput : Bool;
      bAtSetpoint : Bool;
   END_VAR

   VAR_IN_OUT 
      sTag : "stOnOffRegulator";
   END_VAR

   VAR 
      Controller { S7_SetPoint := 'False'} : "fbHysteresis";
   END_VAR

   VAR_TEMP 
      fSetpoint : Real;
      Enabled : Bool;
   END_VAR


BEGIN
	// 1-sided on/off controller
	// Above = 1: regulate when Process Value (PV) above threshold. Eg. cooling, emptying, depressurizing
	// Above = 0: regulate when PV below threshold. Eg. heating, filling, pressurizing
	
	// Reset manual modes.
	IF #bReset THEN
	    #sTag.bManualMode := FALSE;
	    #sTag.fManualSetpoint := 0.0;
	    #sTag.bManualOverride := FALSE;
	    #sTag.bOverrideCmd := FALSE;
	END_IF;
	
	IF #sTag.bManualOverride = TRUE THEN
	    // In manual override, everything is awesome
	    #sTag.bAtSetpoint := TRUE;
	    #sTag.bFault := FALSE;
	    #sTag.bOutput := #sTag.bOverrideCmd;
	ELSE
	    // Choose setpoint
	    IF #sTag.bManualMode = TRUE THEN
	        #fSetpoint := #sTag.fManualSetpoint;
	    ELSE
	        #fSetpoint := #sTag.fSetpoint;
	    END_IF;
	
	    // Enabled when enabled from process and from HMI (Auto), or in Manual mode
	    #Enabled := (#bEnable AND #sTag.bEnable) OR #sTag.bManualMode;
	
	    // Run controller
	    IF #Enabled = TRUE AND #sPV.bError = FALSE THEN
	        #Controller(fValue := #sPV.fValue, fLimit := #fSetpoint, fHysteresis := #sTag.fHysteresis, bType := #Above, bOutput => #sTag.bOutput );
	        #sTag.bAtSetpoint := NOT(#sTag.bOutput);
	    ELSE
	        #sTag.bAtSetpoint := FALSE;
	        #sTag.bOutput  := FALSE;
	    END_IF;
	
	    // Controller fault
	    #sTag.bFault := #sPV.bError;
	
	END_IF;
	
	// Mode
	IF #sTag.bManualOverride = TRUE THEN
	    #sTag.nMode := 3;
	ELSIF #sTag.bManualMode = TRUE THEN
	    #sTag.nMode := 2;
	ELSIF #sTag.bEnable = TRUE THEN
	    #sTag.nMode := 1;
	ELSE
	    #sTag.nMode := 0;
	END_IF;
	
	// Local outputs
	#bOutput := #sTag.bOutput;
	#bAtSetpoint := #sTag.bAtSetpoint;
	
	
END_FUNCTION_BLOCK

FUNCTION_BLOCK "fbPI_Regulator"   // FB21, FBD
TITLE = PI Regulator
{ S7_Optimized_Access := 'TRUE' }
VERSION : 0.1
// stored: AutoNumber true, IsIECCheckEnabled false, IsRetainMemResEnabled false, MemoryReserve 0, SetENOAutomatically false, UDAEnableTagReadback false
   VAR_INPUT
      sPV : "stCalcValue";   // Process value
      fCycleTime : Real;
      bEnable : Bool;
      bReset : Bool;
   END_VAR
   VAR_OUTPUT
      fOut : Real;
      bAtMin : Bool;
      bAtMax : Bool;
   END_VAR
   VAR_IN_OUT
      sTag : "stPI_Regulator";
   END_VAR
   VAR
      D_Mem : Real;
      I_Mem : Real;
      Param_Mem : Real;
   END_VAR
   VAR_TEMP
      Enabled : Bool;
      fDeviation : Real;
   END_VAR
BEGIN

REGION Network 1: Reset manual mode
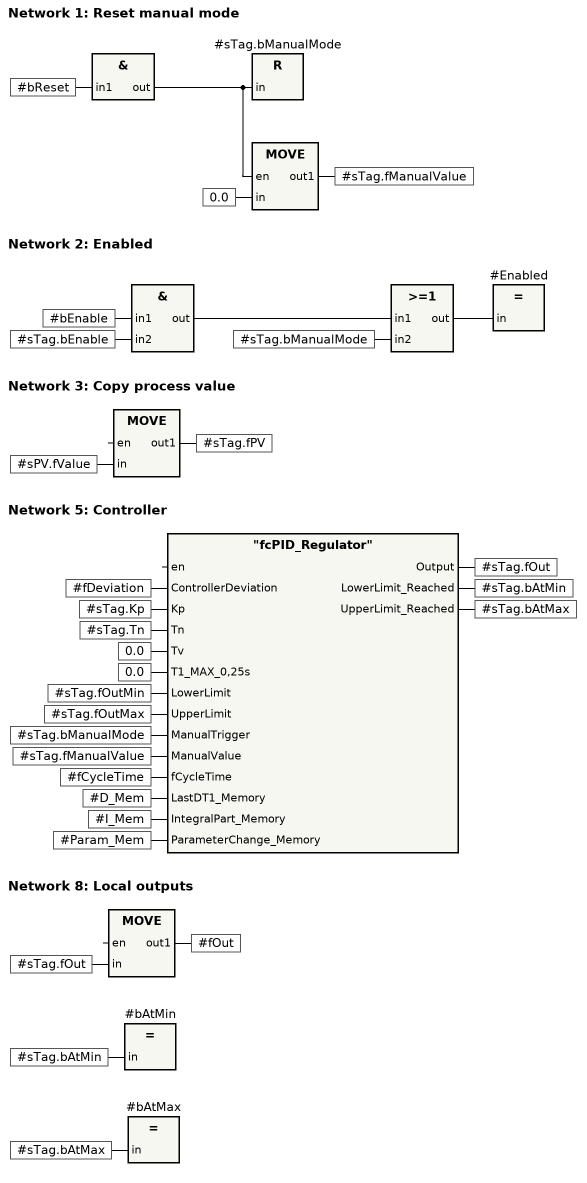
   IF #bReset THEN
       #sTag.bManualMode := FALSE;
       #sTag.fManualValue := 0.0;
   END_IF;
END_REGION

REGION Network 2: Enabled
   // Local input is from process control logic: when to run the regulator
   // Tag input is from HMI: do we want to run this regulator at all
   #Enabled := (#bEnable AND #sTag.bEnable) OR #sTag.bManualMode;
END_REGION

REGION Network 3: Copy process value
   #sTag.fPV := #sPV.fValue;
END_REGION

REGION Network 4 (SCL): Deviation
   // NaN detection
   IF "isNaN"(#sTag.fSP) OR "isNaN"(#sTag.fPV) THEN
       #fDeviation := 0.0;
       #sTag.bFault := TRUE;
   ELSE
       #fDeviation := #sTag.fSP - #sTag.fPV;
       #sTag.bFault := FALSE;
   END_IF;
END_REGION

REGION Network 5: Controller
   // NOTE: controller always runs regardless of mode
   "fcPID_Regulator"(ControllerDeviation := #fDeviation,
                     Kp := #sTag.Kp,
                     Tn := #sTag.Tn,
                     Tv := 0.0,
                     "T1_MAX_0,25s" := 0.0,
                     LowerLimit := #sTag.fOutMin,
                     UpperLimit := #sTag.fOutMax,
                     ManualTrigger := #sTag.bManualMode,
                     ManualValue := #sTag.fManualValue,
                     fCycleTime := #fCycleTime,
                     LastDT1_Memory := #D_Mem,
                     IntegralPart_Memory := #I_Mem,
                     ParameterChange_Memory := #Param_Mem,
                     Output => #sTag.fOut,
                     LowerLimit_Reached => #sTag.bAtMin,
                     UpperLimit_Reached => #sTag.bAtMax);
END_REGION

REGION Network 6 (SCL): Disable
   IF #Enabled = FALSE OR #sTag.bFault = TRUE THEN
       #sTag.fOut := 0.0;
       #sTag.bAtMin := FALSE;
       #sTag.bAtMax := FALSE;
   END_IF;
END_REGION

REGION Network 7 (SCL): Mode
   // Mode
   IF #sTag.bManualMode = TRUE THEN
       #sTag.nMode := 2;
   ELSIF #sTag.bEnable = TRUE THEN
       #sTag.nMode := 1;
   ELSE
       #sTag.nMode := 0;
   END_IF;
END_REGION

REGION Network 8: Local outputs
   #fOut := #sTag.fOut;
   #bAtMin := #sTag.bAtMin;
   #bAtMax := #sTag.bAtMax;
END_REGION
END_FUNCTION_BLOCK

FUNCTION_BLOCK "CrankcasePressureControl"   // FB2, FBD
TITLE = Crankcase pressure control system (CPC)
{ S7_Optimized_Access := 'TRUE' }
VERSION : 0.1
// stored: AutoNumber true, IsIECCheckEnabled false, IsRetainMemResEnabled false, MemoryReserve 100, SetENOAutomatically false, UDAEnableTagReadback false
   VAR_INPUT
      bEnable { ExternalAccessible := 'False'; ExternalVisible := 'False'; ExternalWritable := 'False'} : Bool;
      bReset { ExternalAccessible := 'False'; ExternalVisible := 'False'; ExternalWritable := 'False'} : Bool;   // 1 = reset manual modes
   END_VAR
   VAR_OUTPUT
      bPumpOut { ExternalAccessible := 'False'; ExternalVisible := 'False'; ExternalWritable := 'False'} : Bool;   // 1 = run pump, 0 = do not run pump
   END_VAR
   VAR
      Cooler { ExternalAccessible := 'False'; ExternalVisible := 'False'; ExternalWritable := 'False'; S7_SetPoint := 'True'} : "fbPI_Regulator";
      LevelControl { ExternalAccessible := 'False'; ExternalVisible := 'False'; ExternalWritable := 'False'; S7_SetPoint := 'True'} : "fbOnOffRegulator";   // Regulate level based on direct level measurement
      LevelControl2 { ExternalAccessible := 'False'; ExternalVisible := 'False'; ExternalWritable := 'False'; S7_SetPoint := 'True'} : "fbProgressivePeriodicRegulator4";
      HighAlarm { ExternalAccessible := 'False'; ExternalVisible := 'False'; ExternalWritable := 'False'; S7_SetPoint := 'True'} : "fbHighAlarm";
   END_VAR
   VAR_TEMP
      bPumpOut1 : Bool;
      bPumpOut2 : Bool;
   END_VAR
BEGIN

REGION Network 1: Cooling fan regulator
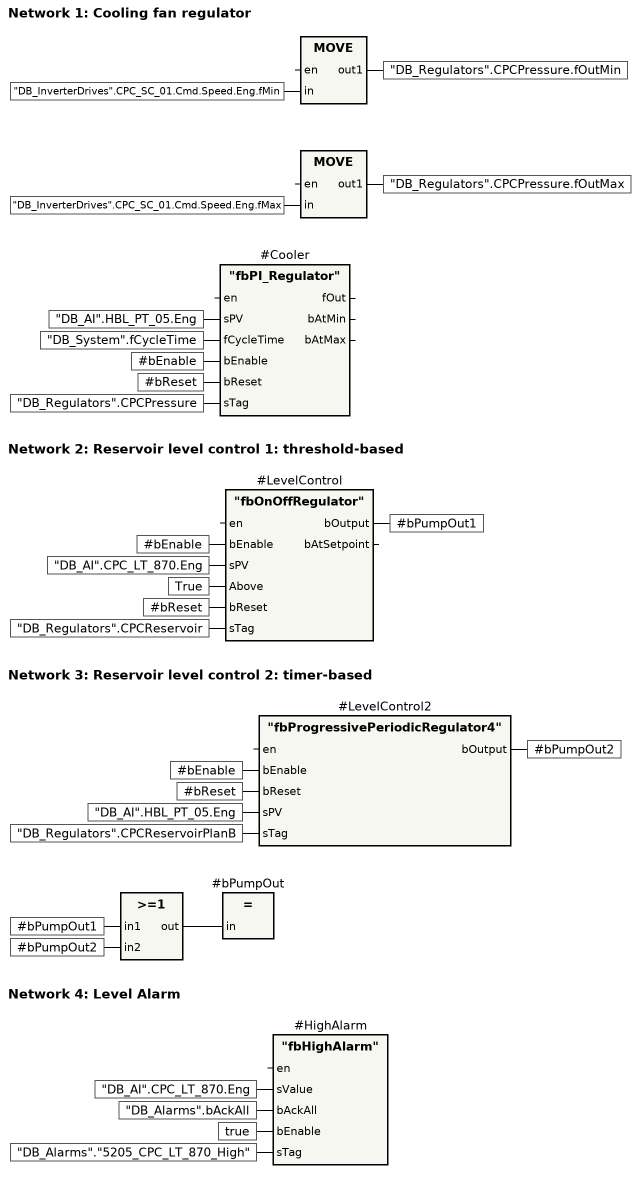
   "DB_Regulators".CPCPressure.fOutMin := "DB_InverterDrives".CPC_SC_01.Cmd.Speed.Eng.fMin;
   "DB_Regulators".CPCPressure.fOutMax := "DB_InverterDrives".CPC_SC_01.Cmd.Speed.Eng.fMax;
   #Cooler(sPV := "DB_AI".HBL_PT_05.Eng,   // "fbPI_Regulator"
           fCycleTime := "DB_System".fCycleTime,
           bEnable := #bEnable,
           bReset := #bReset,
           sTag := "DB_Regulators".CPCPressure);
END_REGION

REGION Network 2: Reservoir level control 1: threshold-based
   #LevelControl(bEnable := #bEnable,   // "fbOnOffRegulator"
                 sPV := "DB_AI".CPC_LT_870.Eng,
                 Above := True,
                 bReset := #bReset,
                 sTag := "DB_Regulators".CPCReservoir,
                 bOutput => #bPumpOut1);
END_REGION

REGION Network 3: Reservoir level control 2: timer-based
   #LevelControl2(bEnable := #bEnable,   // "fbProgressivePeriodicRegulator4"
                  bReset := #bReset,
                  sPV := "DB_AI".HBL_PT_05.Eng,
                  sTag := "DB_Regulators".CPCReservoirPlanB,
                  bOutput => #bPumpOut2);
   #bPumpOut := #bPumpOut1 OR #bPumpOut2;
END_REGION

REGION Network 4: Level Alarm
   #HighAlarm(sValue := "DB_AI".CPC_LT_870.Eng,   // "fbHighAlarm"
              bAckAll := "DB_Alarms".bAckAll,
              bEnable := true,
              sTag := "DB_Alarms"."5205_CPC_LT_870_High");
END_REGION
END_FUNCTION_BLOCK

FUNCTION_BLOCK "fbProgressivePeriodicRegulator4"
{ S7_Optimized_Access := 'TRUE' }
VERSION : 0.1
   VAR_INPUT 
      bEnable : Bool;   // 1 = enable regulator, 0 = disable regulator
      bReset : Bool;   // 1 = reset everything to zero
      sPV : "stCalcValue";   // Process value
   END_VAR

   VAR_OUTPUT 
      bOutput : Bool;
   END_VAR

   VAR_IN_OUT 
      sTag : "stProgressivePeriodicRegulator4";
   END_VAR

   VAR 
      Controller : "fbPWMController";
   END_VAR

   VAR_TEMP 
      Enabled : Bool;
   END_VAR


BEGIN
	// Progressive periodic regulator (4)
	// Periodic control of an output based on a threshold
	// There is one fixed on-period
	// Auto mode: use a table of thresholds with corresponding periods (4 entries)
	// Manual mode: use a fixed operiod
	// Manual override: force the output on or off
	
	// Copy to tag
	#sTag.fPV := #sPV.fValue;
	
	// Reset manual modes.
	IF #bReset THEN
	    #sTag.bManualMode := FALSE;
	    #sTag.tManualPeriod := T#0s;
	    #sTag.bManualOverride := FALSE;
	    #sTag.bOverrideCmd := FALSE;
	END_IF;
	
	// Controller
	IF #sTag.bManualOverride = TRUE THEN
	    // In manual override, everything is awesome
	    #sTag.bFault := FALSE;
	    #sTag.bOutput := #sTag.bOverrideCmd;
	ELSE
	    // Choose fixed or progressive period
	    IF #sTag.bManualMode = TRUE THEN
	        #sTag.tPeriod := #sTag.tManualPeriod;
	    ELSE
	        IF #sTag.fPV >= #sTag.Param.Limit[0] AND #sTag.fPV < #sTag.Param.Limit[1] THEN
	            #sTag.tPeriod := #sTag.Param.Period[0];
	        ELSIF #sTag.fPV >= #sTag.Param.Limit[1] AND #sTag.fPV < #sTag.Param.Limit[2] THEN
	            #sTag.tPeriod := #sTag.Param.Period[1];
	        ELSIF #sTag.fPV >= #sTag.Param.Limit[2] AND #sTag.fPV < #sTag.Param.Limit[3] THEN
	            #sTag.tPeriod := #sTag.Param.Period[2];
	        ELSIF #sTag.fPV >= #sTag.Param.Limit[3] THEN
	            #sTag.tPeriod := #sTag.Param.Period[3];
	        END_IF;
	    END_IF;
	
	    // Enabled when enabled from process and from HMI (Auto), or in Manual mode
	    #Enabled := (#bEnable AND #sTag.bEnable) OR #sTag.bManualMode;
	
	    // Run controller
	    #Controller(bEnable := #Enabled AND (#sPV.bError = FALSE), 
	                tOnTime := #sTag.tOnTime, 
	                tPeriod := #sTag.tPeriod, 
	                bOut => #sTag.bOutput, 
	                tOnTimeElapsed => #sTag.tOnTimeElapsed, 
	                tPeriodElapsed => #sTag.tPeriodElapsed);
	   
	    // Controller fault
	    #sTag.bFault := #sPV.bError;
	
	END_IF;
	
	// Mode
	IF #sTag.bManualOverride = TRUE THEN
	    #sTag.nMode := 3;
	ELSIF #sTag.bManualMode = TRUE THEN
	    #sTag.nMode := 2;
	ELSIF #sTag.bEnable = TRUE THEN
	    #sTag.nMode := 1;
	ELSE
	    #sTag.nMode := 0;
	END_IF;
	
	// Local outputs
	#bOutput := #sTag.bOutput;
END_FUNCTION_BLOCK

FUNCTION_BLOCK "fbPWMController"   // FB35, FBD
TITLE = PWM Controller
{ S7_Optimized_Access := 'TRUE' }
VERSION : 0.1
// stored: AutoNumber true, IsIECCheckEnabled false, IsRetainMemResEnabled false, MemoryReserve 0, SetENOAutomatically false, UDAEnableTagReadback false
   VAR_INPUT
      bEnable : Bool;   // 1 = enable controller, 0 = disable
      tOnTime : Time;
      tPeriod : Time;
   END_VAR
   VAR_OUTPUT
      bOut : Bool;
      tOnTimeElapsed : Time;
      tPeriodElapsed : Time;
   END_VAR
   VAR
      PeriodTimer { S7_SetPoint := 'True'} : TP_TIME;
      OnTimer : TP_TIME;
      bOnTime { S7_SetPoint := 'True'} : Bool := True;
   END_VAR
BEGIN

REGION Network 1: Trigger the output
   // Note: if output should start LOW, set initial value of bOnTime to FALSE
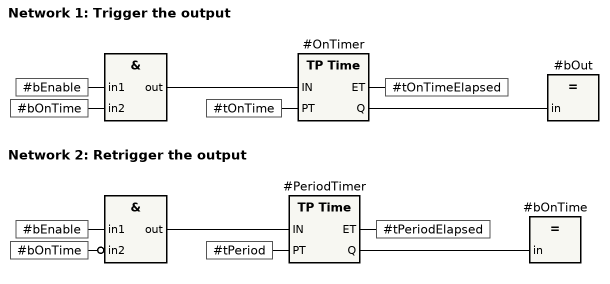
   #OnTimer(IN := #bEnable AND #bOnTime, PT := #tOnTime, ET => #tOnTimeElapsed);   // TP
   #bOut := #OnTimer.Q;
END_REGION

REGION Network 2: Retrigger the output
   #PeriodTimer(IN := #bEnable AND NOT #bOnTime, PT := #tPeriod, ET => #tPeriodElapsed);   // TP
   #bOnTime := #PeriodTimer.Q;
END_REGION

REGION Network 3 (SCL): Reset
   IF #bEnable = FALSE THEN
       RESET_TIMER(#PeriodTimer);
       RESET_TIMER(#OnTimer);
   END_IF;
END_REGION
END_FUNCTION_BLOCK

FUNCTION_BLOCK "OilSeparator"   // FB15, FBD
TITLE = Oil Separator
{ S7_Optimized_Access := 'TRUE' }
VERSION : 0.1
// stored: AutoNumber true, IsIECCheckEnabled false, IsRetainMemResEnabled false, MemoryReserve 100, SetENOAutomatically false, UDAEnableTagReadback false
   VAR_INPUT
      bEnable { ExternalAccessible := 'False'; ExternalVisible := 'False'; ExternalWritable := 'False'} : Bool;
      bReset { ExternalAccessible := 'False'; ExternalVisible := 'False'; ExternalWritable := 'False'} : Bool;   // 1 = reset manual modes
   END_VAR
   VAR
      Regulator { ExternalAccessible := 'False'; ExternalVisible := 'False'; ExternalWritable := 'False'} : "fbOnOffRegulator";
      Alarm { ExternalAccessible := 'False'; ExternalVisible := 'False'; ExternalWritable := 'False'; S7_SetPoint := 'True'} : "fbDigitalAlarm";
      Stage1 { S7_SetPoint := 'True'} : "fbOnOffRegulator2";
      Stage2 { S7_SetPoint := 'True'} : "fbOnOffRegulator2";
   END_VAR
   VAR_TEMP
      Enabled : Bool;
   END_VAR
BEGIN

REGION Network 1: Stage 1 level control
   // Run only when the pressure in oil separator Stage 1 is greater than the oil sump, so oil will move from oil separator to sump
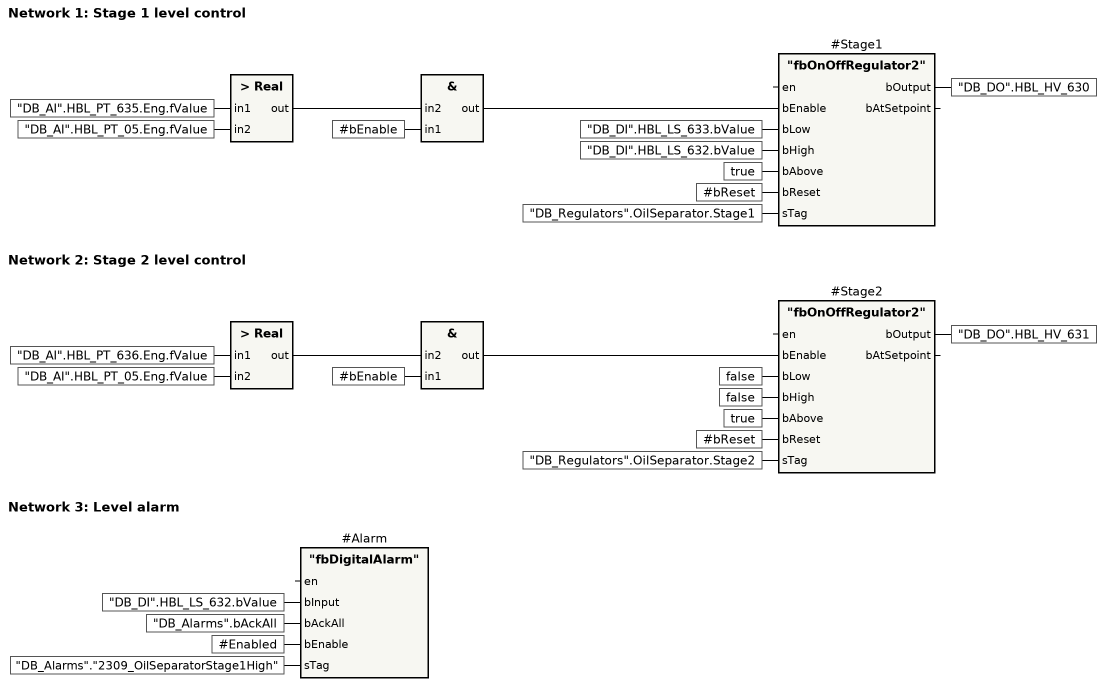
   #Stage1(bEnable := ("DB_AI".HBL_PT_635.Eng.fValue > "DB_AI".HBL_PT_05.Eng.fValue) AND #bEnable,   // "fbOnOffRegulator2"
           bLow := "DB_DI".HBL_LS_633.bValue,
           bHigh := "DB_DI".HBL_LS_632.bValue,
           bAbove := true,
           bReset := #bReset,
           sTag := "DB_Regulators".OilSeparator.Stage1,
           bOutput => "DB_DO".HBL_HV_630);
END_REGION

REGION Network 2: Stage 2 level control
   // Run only when the pressure in oil separator Stage 2 is greater than the oil sump, so oil will move from oil separator to sump
   // 10.02.2025 TSS: Currently no level switches in the P&ID, not sure of the control strategy
   #Stage2(bEnable := ("DB_AI".HBL_PT_636.Eng.fValue > "DB_AI".HBL_PT_05.Eng.fValue) AND #bEnable,   // "fbOnOffRegulator2"
           bLow := false,
           bHigh := false,
           bAbove := true,
           bReset := #bReset,
           sTag := "DB_Regulators".OilSeparator.Stage2,
           bOutput => "DB_DO".HBL_HV_631);
END_REGION

REGION Network 3: Level alarm
   // High level for a long time is probably worth knowing about
   #Alarm(bInput := "DB_DI".HBL_LS_632.bValue,   // "fbDigitalAlarm"
          bAckAll := "DB_Alarms".bAckAll,
          bEnable := #Enabled,
          sTag := "DB_Alarms"."2309_OilSeparatorStage1High");
END_REGION
END_FUNCTION_BLOCK

FUNCTION_BLOCK "fbOnOffRegulator2"
{ S7_Optimized_Access := 'TRUE' }
VERSION : 0.1
   VAR_INPUT 
      bEnable : Bool;   // Enable from process. 1 = enabled, 0 = disabled
      bLow : Bool;   // Lower level switch (1 = level is above switch, 0 = level is below switch)
      bHigh : Bool;   // Higher level switch (1 = level is above switch, 0 = level is below switch)
      bAbove : Bool;   // 1 = regulate when above threshold, 0 = regulate when below threshold
      bReset : Bool;   // 1 = reset manual modes
   END_VAR

   VAR_OUTPUT 
      bOutput : Bool;
      bAtSetpoint : Bool;
   END_VAR

   VAR_IN_OUT 
      sTag : "stOnOffRegulator2";
   END_VAR

   VAR 
      Controller { S7_SetPoint := 'False'} : "fbHysteresis2";
   END_VAR

   VAR_TEMP 
      fSetpoint : Real;
      Enabled : Bool;
   END_VAR


BEGIN
	// 1-sided on/off controller with switch inputs
	// Above = 1: regulate when Process Value (PV) above threshold. Eg. cooling, emptying, depressurizing
	// Above = 0: regulate when PV below threshold. Eg. heating, filling, pressurizing
	
	// Reset manual modes.
	IF #bReset THEN
	    #sTag.bManualOverride := FALSE;
	    #sTag.bOverrideCmd := FALSE;
	END_IF;
	
	IF #sTag.bManualOverride = TRUE THEN
	    // In manual override, everything is awesome
	    #sTag.bFault := FALSE;
	    #sTag.bOutput := #sTag.bOverrideCmd;
	    #sTag.bAtSetpoint := NOT(#sTag.bOutput);
	ELSE
	
	    // Enabled when enabled from process and from HMI (Auto)
	    #Enabled := (#bEnable AND #sTag.bEnable);
	
	    // Run controller
	    #Controller(bEnable := #Enabled, bLow := #bLow, bHigh := #bHigh, bReset := #bReset, bAbove := #bAbove, bOut => #sTag.bOutput );
	
